C01824=1209.441,-97.315,-38.143,179.366,5.454,149.145
C01825=1209.446,-97.564,-38.133,179.364,5.455,149.146
C01826=1209.452,-97.814,-38.123,179.362,5.454,149.146
C01827=1209.457,-98.064,-38.112,179.360,5.454,149.147
C01828=1209.462,-98.314,-38.102,179.357,5.454,149.148
C01829=1209.467,-98.564,-38.092,179.355,5.454,149.149
C01830=1209.472,-98.813,-38.082,179.353,5.454,149.149
C01831=1209.478,-99.063,-38.071,179.351,5.454,149.150
C01832=1209.483,-99.313,-38.061,179.348,5.453,149.150
C01833=1209.488,-99.562,-38.051,179.346,5.454,149.151
C01834=1209.493,-99.812,-38.041,179.343,5.453,149.152
C01835=1209.498,-100.062,-38.031,179.342,5.453,149.152
C01836=1209.504,-100.311,-38.020,179.339,5.453,149.153
C01837=1209.510,-100.561,-38.010,179.337,5.453,149.154
C01838=1209.515,-100.832,-37.999,179.334,5.453,149.155
C01839=1209.521,-101.104,-37.988,179.331,5.453,149.155
C01840=1209.526,-101.375,-37.977,179.329,5.453,149.156
C01841=1209.532,-101.646,-37.966,179.327,5.453,149.157
C01842=1209.537,-101.896,-37.956,179.325,5.453,149.157
C01843=1209.542,-102.146,-37.945,179.322,5.452,149.158
C01844=1209.548,-102.395,-37.935,179.320,5.452,149.159
C01845=1209.553,-102.645,-37.925,179.318,5.452,149.159
C01846=1209.558,-102.895,-37.915,179.315,5.452,149.160
C01847=1209.564,-103.145,-37.905,179.313,5.452,149.161
C01848=1209.569,-103.395,-37.895,179.311,5.452,149.161
C01849=1209.574,-103.645,-37.885,179.309,5.452,149.162
C01850=1209.579,-103.894,-37.875,179.306,5.452,149.163
C01851=1209.585,-104.143,-37.865,179.304,5.452,149.163
C01852=1209.590,-104.394,-37.854,179.302,5.452,149.164
C01853=1209.594,-104.643,-37.845,179.299,5.451,149.165
C01854=1209.600,-104.892,-37.834,179.297,5.452,149.165
C01855=1209.605,-105.143,-37.825,179.295,5.451,149.166
C01856=1209.611,-105.393,-37.814,179.293,5.451,149.167
C01857=1209.616,-105.642,-37.805,179.290,5.451,149.167
C01858=1209.621,-105.892,-37.795,179.288,5.451,149.168
C01859=1209.626,-106.142,-37.784,179.286,5.451,149.169
C01860=1209.631,-106.391,-37.774,179.284,5.451,149.169
C01861=1209.637,-106.641,-37.765,179.281,5.450,149.170
C01862=1209.642,-106.891,-37.754,179.279,5.451,149.171
C01863=1209.647,-107.141,-37.745,179.277,5.450,149.171
C01864=1209.653,-107.390,-37.734,179.275,5.451,149.172
C01865=1209.658,-107.640,-37.724,179.272,5.450,149.172
C01866=1209.663,-107.890,-37.715,179.270,5.450,149.173
C01867=1209.668,-108.140,-37.705,179.268,5.450,149.174
C01868=1209.674,-108.389,-37.695,179.265,5.450,149.175
C01869=1209.679,-108.639,-37.685,179.263,5.449,149.175
C01870=1209.684,-108.889,-37.675,179.261,5.450,149.176
C01871=1209.689,-109.139,-37.665,179.259,5.449,149.176
C01872=1209.695,-109.388,-37.655,179.256,5.450,149.177
C01873=1209.700,-109.638,-37.645,179.254,5.449,149.178
C01874=1209.705,-109.888,-37.636,179.252,5.449,149.178
C01875=1209.710,-110.138,-37.626,179.249,5.449,149.179
C01876=1209.716,-110.387,-37.615,179.247,5.449,149.180
C01877=1209.721,-110.637,-37.606,179.245,5.448,149.180
C01878=1209.727,-110.887,-37.596,179.243,5.449,149.181
C01879=1209.732,-111.136,-37.587,179.240,5.448,149.182
C01880=1209.737,-111.386,-37.576,179.238,5.449,149.182
C01881=1209.743,-111.636,-37.567,179.236,5.448,149.183
C01882=1209.747,-111.886,-37.557,179.234,5.448,149.184
C01883=1209.753,-112.135,-37.547,179.231,5.448,149.184
C01884=1209.758,-112.385,-37.538,179.229,5.448,149.185
C01885=1209.763,-112.635,-37.527,179.228,5.448,149.186
C01886=1209.768,-112.885,-37.518,179.225,5.448,149.186
C01887=1209.774,-113.135,-37.508,179.223,5.448,149.187
C01888=1209.780,-113.384,-37.498,179.220,5.448,149.188
C01889=1209.785,-113.634,-37.489,179.219,5.448,149.188
C01890=1209.790,-113.884,-37.479,179.216,5.448,149.189
C01891=1209.795,-114.134,-37.469,179.214,5.448,149.190
C01892=1209.800,-114.384,-37.459,179.212,5.447,149.190
C01893=1209.805,-114.633,-37.450,179.210,5.448,149.191
C01894=1209.811,-114.883,-37.440,179.207,5.447,149.192
C01895=1209.816,-115.132,-37.431,179.205,5.448,149.192
C01896=1209.822,-115.382,-37.420,179.203,5.447,149.193
C01897=1209.826,-115.633,-37.411,179.201,5.447,149.193
C01898=1209.832,-115.882,-37.401,179.198,5.447,149.194
C01899=1209.837,-116.132,-37.392,179.196,5.447,149.195
C01900=1209.843,-116.381,-37.382,179.194,5.446,149.195
C01901=1209.848,-116.631,-37.373,179.192,5.447,149.196
C01902=1209.853,-116.881,-37.363,179.189,5.446,149.197
C01903=1209.858,-117.130,-37.353,179.187,5.446,149.197
C01904=1209.864,-117.381,-37.343,179.185,5.446,149.198
C01905=1209.868,-117.630,-37.334,179.182,5.446,149.199
C01906=1209.874,-117.880,-37.324,179.180,5.447,149.199
C01907=1209.879,-118.130,-37.315,179.178,5.446,149.200
C01908=1209.885,-118.380,-37.305,179.176,5.446,149.201
C01909=1209.890,-118.629,-37.296,179.173,5.446,149.201
C01910=1209.895,-118.879,-37.287,179.172,5.446,149.202
C01911=1209.901,-119.128,-37.276,179.169,5.445,149.203
C01912=1209.906,-119.378,-37.268,179.167,5.446,149.203
C01913=1209.911,-119.628,-37.257,179.164,5.445,149.204
C01914=1209.916,-119.878,-37.248,179.163,5.445,149.204
C01915=1209.922,-120.128,-37.239,179.160,5.445,149.205
C01916=1209.927,-120.378,-37.229,179.158,5.445,149.206
C01917=1209.932,-120.628,-37.220,179.156,5.445,149.206
C01918=1209.938,-120.877,-37.210,179.154,5.445,149.207
C01919=1209.943,-121.127,-37.201,179.151,5.445,149.208
C01920=1209.948,-121.376,-37.191,179.149,5.445,149.208
C01921=1209.953,-121.626,-37.182,179.147,5.445,149.209
C01922=1209.959,-121.876,-37.173,179.145,5.445,149.210
C01923=1209.964,-122.126,-37.163,179.143,5.445,149.210
C01924=1209.969,-122.376,-37.154,179.140,5.444,149.211
C01925=1209.974,-122.625,-37.144,179.138,5.445,149.212
C01926=1209.980,-122.875,-37.135,179.136,5.444,149.212
C01927=1209.985,-123.126,-37.125,179.134,5.444,149.213
C01928=1209.990,-123.375,-37.115,179.131,5.444,149.214
C01929=1209.996,-123.625,-37.106,179.129,5.444,149.214
C01930=1210.000,-123.874,-37.097,179.127,5.443,149.215
C01931=1210.006,-124.124,-37.087,179.125,5.444,149.216
C01932=1210.011,-124.374,-37.078,179.122,5.443,149.216
C01933=1210.016,-124.623,-37.069,179.121,5.443,149.217
C01934=1210.022,-124.874,-37.059,179.119,5.444,149.217
C01935=1210.027,-125.123,-37.050,179.116,5.443,149.218
C01936=1210.032,-125.373,-37.041,179.114,5.444,149.219
C01937=1210.038,-125.623,-37.031,179.112,5.443,149.219
C01938=1210.043,-125.873,-37.022,179.110,5.443,149.220
C01939=1210.048,-126.123,-37.013,179.107,5.443,149.221
C01940=1210.054,-126.372,-37.003,179.105,5.443,149.221
C01941=1210.059,-126.622,-36.994,179.103,5.443,149.222
C01942=1209.638,-126.632,-37.032,179.099,5.446,149.224
C01943=1209.632,-126.382,-37.041,179.101,5.447,149.223
C01944=1209.628,-126.133,-37.051,179.103,5.446,149.223
C01945=1209.622,-125.883,-37.060,179.106,5.447,149.222
C01946=1209.617,-125.633,-37.069,179.107,5.447,149.221
C01947=1209.611,-125.383,-37.078,179.110,5.447,149.221
C01948=1209.606,-125.134,-37.088,179.112,5.447,149.220
C01949=1209.601,-124.884,-37.097,179.114,5.447,149.220
C01950=1209.595,-124.634,-37.106,179.116,5.447,149.219
C01951=1209.590,-124.385,-37.116,179.118,5.447,149.218
C01952=1209.585,-124.135,-37.125,179.121,5.447,149.218
C01953=1209.580,-123.885,-37.134,179.123,5.447,149.217
C01954=1209.574,-123.635,-37.144,179.125,5.447,149.216
C01955=1209.569,-123.385,-37.153,179.127,5.447,149.215
C01956=1209.564,-123.136,-37.162,179.130,5.448,149.215
C01957=1209.558,-122.886,-37.172,179.132,5.447,149.214
C01958=1209.553,-122.636,-37.181,179.134,5.448,149.214
C01959=1209.548,-122.387,-37.191,179.136,5.448,149.213
C01960=1209.542,-122.137,-37.200,179.139,5.448,149.212
C01961=1209.537,-121.887,-37.209,179.141,5.448,149.212
C01962=1209.532,-121.638,-37.219,179.143,5.449,149.211
C01963=1209.526,-121.388,-37.228,179.145,5.448,149.210
C01964=1209.521,-121.138,-37.238,179.147,5.448,149.210
C01965=1209.516,-120.887,-37.248,179.149,5.449,149.209
C01966=1209.511,-120.638,-37.257,179.151,5.448,149.209
C01967=1209.506,-120.388,-37.266,179.154,5.449,149.208
C01968=1209.500,-120.138,-37.276,179.156,5.448,149.207
C01969=1209.495,-119.889,-37.285,179.158,5.449,149.207
C01970=1209.489,-119.639,-37.295,179.160,5.449,149.206
C01971=1209.484,-119.390,-37.305,179.163,5.449,149.205
C01972=1209.479,-119.139,-37.314,179.165,5.449,149.205
C01973=1209.474,-118.890,-37.324,179.167,5.449,149.204
C01974=1209.468,-118.640,-37.333,179.169,5.449,149.203
C01975=1209.463,-118.391,-37.343,179.172,5.449,149.203
C01976=1209.458,-118.140,-37.352,179.174,5.449,149.202
C01977=1209.453,-117.891,-37.362,179.176,5.450,149.201
C01978=1209.448,-117.641,-37.371,179.179,5.449,149.201
C01979=1209.442,-117.391,-37.381,179.180,5.449,149.200
C01980=1209.437,-117.141,-37.390,179.183,5.450,149.199
C01981=1209.431,-116.892,-37.400,179.185,5.449,149.199
C01982=1209.426,-116.642,-37.409,179.188,5.450,149.198
C01983=1209.420,-116.392,-37.420,179.189,5.450,149.197
C01984=1209.416,-116.142,-37.429,179.192,5.450,149.197
C01985=1209.410,-115.892,-37.439,179.194,5.450,149.196
C01986=1209.405,-115.643,-37.448,179.196,5.451,149.196
C01987=1209.399,-115.393,-37.458,179.198,5.450,149.195
C01988=1209.395,-115.144,-37.468,179.201,5.451,149.194
C01989=1209.389,-114.894,-37.477,179.203,5.450,149.193
C01990=1209.384,-114.644,-37.487,179.205,5.451,149.193
C01991=1209.379,-114.394,-37.497,179.207,5.451,149.192
C01992=1209.374,-114.144,-37.506,179.210,5.451,149.191
C01993=1209.368,-113.895,-37.517,179.212,5.451,149.191
C01994=1209.363,-113.645,-37.525,179.214,5.452,149.190
C01995=1209.357,-113.395,-37.536,179.216,5.451,149.190
C01996=1209.352,-113.145,-37.545,179.219,5.452,149.189
C01997=1209.347,-112.895,-37.555,179.221,5.452,149.188
C01998=1209.342,-112.646,-37.565,179.223,5.452,149.188
C01999=1209.336,-112.396,-37.574,179.225,5.452,149.187
C02000=1209.331,-112.146,-37.584,179.228,5.452,149.186
C02001=1209.326,-111.897,-37.594,179.230,5.452,149.186
C02002=1209.320,-111.647,-37.604,179.232,5.452,149.185
C02003=1209.316,-111.397,-37.614,179.234,5.452,149.184
C02004=1209.310,-111.147,-37.624,179.237,5.452,149.184
C02005=1209.305,-110.898,-37.633,179.239,5.452,149.183
C02006=1209.299,-110.648,-37.643,179.241,5.452,149.182
C02007=1209.294,-110.399,-37.653,179.243,5.452,149.182
C02008=1209.289,-110.148,-37.662,179.245,5.452,149.181
C02009=1209.284,-109.898,-37.673,179.248,5.453,149.181
C02010=1209.279,-109.649,-37.682,179.250,5.452,149.180
C02011=1209.273,-109.400,-37.692,179.253,5.453,149.179
C02012=1209.268,-109.149,-37.702,179.254,5.453,149.179
C02013=1209.263,-108.900,-37.712,179.257,5.453,149.178
C02014=1209.257,-108.650,-37.722,179.259,5.453,149.177
C02015=1209.252,-108.400,-37.732,179.262,5.453,149.176
C02016=1209.247,-108.151,-37.741,179.263,5.453,149.176
C02017=1209.242,-107.900,-37.752,179.266,5.454,149.175
C02018=1209.236,-107.651,-37.762,179.268,5.453,149.175
C02019=1209.231,-107.402,-37.772,179.271,5.454,149.174
C02020=1209.225,-107.151,-37.781,179.272,5.454,149.173
C02021=1209.220,-106.901,-37.792,179.275,5.454,149.173
C02022=1209.215,-106.652,-37.801,179.277,5.454,149.172
C02023=1209.210,-106.402,-37.811,179.280,5.454,149.171
C02024=1209.205,-106.152,-37.822,179.281,5.454,149.171
C02025=1209.200,-105.902,-37.831,179.284,5.455,149.170
C02026=1209.194,-105.653,-37.841,179.286,5.454,149.169
C02027=1209.189,-105.403,-37.851,179.289,5.455,149.169
C02028=1209.184,-105.153,-37.861,179.291,5.454,149.168
C02029=1209.179,-104.904,-37.872,179.293,5.455,149.167
C02030=1209.173,-104.654,-37.882,179.295,5.455,149.167
C02031=1209.168,-104.405,-37.891,179.298,5.455,149.166
C02032=1209.163,-104.154,-37.901,179.300,5.455,149.165
C02033=1209.157,-103.905,-37.911,179.302,5.456,149.165
C02034=1209.152,-103.655,-37.922,179.304,5.455,149.164
C02035=1209.147,-103.405,-37.932,179.307,5.456,149.163
C02036=1209.142,-103.156,-37.942,179.309,5.455,149.163
C02037=1209.136,-102.906,-37.952,179.311,5.456,149.162
C02038=1209.132,-102.656,-37.962,179.313,5.456,149.161
C02039=1209.126,-102.407,-37.972,179.316,5.456,149.161
C02040=1209.121,-102.157,-37.982,179.318,5.456,149.160
C02041=1209.115,-101.906,-37.992,179.320,5.456,149.159
C02042=1209.111,-101.657,-38.002,179.322,5.456,149.159
C02043=1209.105,-101.385,-38.013,179.325,5.456,149.158
C02044=1209.099,-101.115,-38.024,179.328,5.457,149.157
C02045=1209.093,-100.843,-38.036,179.330,5.457,149.157
C02046=1209.088,-100.572,-38.046,179.332,5.457,149.156
C02047=1209.082,-100.322,-38.057,179.334,5.457,149.155
C02048=1209.077,-100.073,-38.067,179.337,5.457,149.154
C02049=1209.072,-99.822,-38.077,179.339,5.457,149.154
C02050=1209.067,-99.573,-38.087,179.341,5.457,149.153
C02051=1209.062,-99.323,-38.098,179.343,5.457,149.153
C02052=1209.056,-99.073,-38.108,179.346,5.457,149.152
C02053=1209.051,-98.824,-38.118,179.348,5.457,149.151
C02054=1209.046,-98.574,-38.129,179.351,5.457,149.150
C02055=1209.041,-98.324,-38.138,179.352,5.457,149.150
C02056=1209.035,-98.075,-38.148,179.355,5.458,149.149
C02057=1209.030,-97.825,-38.159,179.357,5.458,149.149
C02058=1209.024,-97.575,-38.169,179.360,5.458,149.148
C02059=1209.019,-97.326,-38.179,179.361,5.458,149.147
C02060=1209.014,-97.075,-38.190,179.364,5.458,149.147
C02061=1209.008,-96.826,-38.200,179.366,5.458,149.146
C02062=1209.004,-96.576,-38.210,179.369,5.458,149.145
C02063=1208.999,-96.327,-38.221,179.372,5.459,149.144
C02064=1208.993,-96.077,-38.231,179.373,5.459,149.144
C02065=1208.988,-95.827,-38.242,179.376,5.459,149.143
C02066=1208.983,-95.578,-38.252,179.378,5.459,149.143
C02067=1208.978,-95.327,-38.263,179.381,5.459,149.142
C02068=1208.972,-95.078,-38.273,179.383,5.459,149.141
C02069=1208.966,-94.828,-38.283,179.385,5.460,149.141
C02070=1208.961,-94.578,-38.294,179.387,5.459,149.140
C02071=1208.956,-94.328,-38.304,179.390,5.460,149.139
C02072=1208.952,-94.079,-38.315,179.392,5.459,149.139
C02073=1208.946,-93.830,-38.325,179.394,5.460,149.138
C02074=1208.941,-93.579,-38.335,179.396,5.460,149.137
C02075=1208.936,-93.330,-38.346,179.399,5.460,149.137
C02076=1208.930,-93.080,-38.356,179.401,5.460,149.136
C02077=1208.925,-92.830,-38.366,179.403,5.460,149.135
C02078=1208.919,-92.580,-38.377,179.406,5.460,149.135
C02079=1208.915,-92.331,-38.388,179.408,5.461,149.134
C02080=1208.909,-92.081,-38.398,179.410,5.460,149.133
C02081=1208.904,-91.831,-38.409,179.413,5.461,149.133
C02082=1208.899,-91.581,-38.419,179.415,5.460,149.132
C02083=1208.894,-91.331,-38.429,179.417,5.461,149.131
C02084=1208.888,-91.082,-38.440,179.419,5.462,149.131
C02085=1208.883,-90.833,-38.451,179.422,5.461,149.130
C02086=1208.878,-90.583,-38.461,179.424,5.462,149.129
C02087=1208.872,-90.333,-38.471,179.426,5.461,149.129
C02088=1208.867,-90.083,-38.483,179.429,5.462,149.128
C02089=1208.862,-89.834,-38.493,179.431,5.462,149.127
C02090=1208.857,-89.584,-38.503,179.433,5.462,149.127
C02091=1208.851,-89.334,-38.514,179.435,5.462,149.126
C02092=1208.846,-89.084,-38.525,179.438,5.462,149.125
C02093=1208.841,-88.835,-38.535,179.440,5.462,149.125
C02094=1208.836,-88.585,-38.546,179.442,5.463,149.124
C02095=1208.831,-88.336,-38.557,179.444,5.462,149.123
C02096=1208.826,-88.085,-38.567,179.447,5.463,149.123
C02097=1208.820,-87.836,-38.577,179.449,5.462,149.122
C02098=1208.815,-87.586,-38.589,179.452,5.463,149.121
C02099=1208.810,-87.337,-38.599,179.454,5.463,149.120
C02100=1208.805,-87.086,-38.609,179.456,5.463,149.120
C02101=1208.799,-86.837,-38.620,179.459,5.464,149.119
C02102=1208.794,-86.587,-38.631,179.461,5.463,149.119
C02103=1208.789,-86.338,-38.641,179.464,5.464,149.118
C02104=1208.784,-86.088,-38.652,179.466,5.463,149.117
C02105=1208.779,-85.838,-38.663,179.468,5.464,149.117
C02106=1208.774,-85.588,-38.673,179.470,5.464,149.116
C02107=1208.769,-85.339,-38.685,179.473,5.464,149.115
C02108=1208.762,-85.089,-38.695,179.475,5.464,149.115
C02109=1208.757,-84.839,-38.706,179.477,5.464,149.114
C02110=1208.752,-84.590,-38.717,179.479,5.464,149.113
C02111=1208.747,-84.339,-38.727,179.482,5.465,149.113
C02112=1208.742,-84.091,-38.738,179.484,5.465,149.112
C02113=1208.737,-83.840,-38.749,179.486,5.465,149.111
C02114=1208.732,-83.591,-38.760,179.489,5.465,149.111
C02115=1208.727,-83.341,-38.770,179.491,5.465,149.110
C02116=1208.722,-83.091,-38.781,179.494,5.465,149.109
C02117=1208.716,-82.842,-38.793,179.495,5.465,149.109
C02118=1208.711,-82.591,-38.803,179.498,5.466,149.108
C02119=1208.705,-82.342,-38.814,179.500,5.465,149.107
C02120=1208.700,-82.092,-38.825,179.503,5.466,149.106
C02121=1208.696,-81.843,-38.836,179.505,5.466,149.106
C02122=1208.690,-81.593,-38.846,179.507,5.466,149.105
C02123=1208.685,-81.343,-38.857,179.510,5.467,149.105
C02124=1208.679,-81.094,-38.868,179.512,5.466,149.104
C02125=1208.674,-80.844,-38.879,179.515,5.467,149.103
C02126=1208.669,-80.594,-38.890,179.517,5.466,149.102
C02127=1208.664,-80.345,-38.901,179.519,5.467,149.102
C02128=1208.659,-80.095,-38.912,179.521,5.467,149.101
C02129=1208.653,-79.845,-38.923,179.524,5.467,149.101
C02130=1208.648,-79.595,-38.934,179.526,5.468,149.100
C02131=1208.643,-79.345,-38.945,179.528,5.467,149.099
C02132=1208.638,-79.096,-38.955,179.531,5.468,149.098
C02133=1208.633,-78.846,-38.966,179.533,5.467,149.098
C02134=1208.627,-78.597,-38.978,179.535,5.468,149.097
C02135=1208.622,-78.347,-38.989,179.537,5.468,149.097
C02136=1208.617,-78.097,-39.000,179.540,5.468,149.096
C02137=1208.612,-77.848,-39.010,179.542,5.468,149.095
C02138=1208.606,-77.598,-39.022,179.545,5.468,149.094
C02139=1208.601,-77.347,-39.032,179.547,5.469,149.094
C02140=1208.596,-77.099,-39.043,179.549,5.468,149.093
C02141=1208.591,-76.849,-39.055,179.552,5.469,149.093
C02142=1208.586,-76.598,-39.066,179.554,5.469,149.092
C02143=1208.580,-76.349,-39.077,179.556,5.469,149.091
C02144=1208.576,-76.100,-39.088,179.559,5.469,149.090
C02145=1208.570,-75.849,-39.099,179.561,5.469,149.090
C02146=1208.565,-75.600,-39.110,179.564,5.470,149.089
C02147=1208.559,-75.329,-39.122,179.566,5.470,149.088
C02148=1208.554,-75.059,-39.134,179.569,5.470,149.088
C02149=1208.548,-74.788,-39.146,179.571,5.470,149.087
C02150=1208.542,-74.517,-39.158,179.573,5.470,149.086
C02151=1208.537,-74.268,-39.169,179.576,5.470,149.085
C02152=1208.531,-74.018,-39.180,179.579,5.471,149.085
C02153=1208.526,-73.768,-39.192,179.580,5.471,149.084
C02154=1208.522,-73.519,-39.203,179.583,5.471,149.084
C02155=1208.516,-73.269,-39.214,179.585,5.471,149.083
C02156=1208.511,-73.019,-39.225,179.588,5.471,149.082
C02157=1208.506,-72.770,-39.236,179.590,5.471,149.081
C02158=1208.500,-72.520,-39.248,179.593,5.472,149.081
C02159=1208.495,-72.271,-39.259,179.595,5.472,149.080
C02160=1208.490,-72.020,-39.270,179.597,5.472,149.080
C02161=1208.484,-71.771,-39.281,179.599,5.472,149.079
C02162=1208.480,-71.522,-39.292,179.602,5.472,149.078
C02163=1208.475,-71.272,-39.304,179.604,5.473,149.077
C02164=1208.469,-71.021,-39.315,179.607,5.473,149.077
C02165=1208.464,-70.773,-39.326,179.609,5.473,149.076
C02166=1208.458,-70.523,-39.338,179.611,5.473,149.076
C02167=1208.454,-70.273,-39.349,179.613,5.473,149.075
C02168=1208.449,-70.023,-39.360,179.616,5.473,149.074
C02169=1208.443,-69.773,-39.371,179.618,5.473,149.073
C02170=1208.438,-69.524,-39.382,179.621,5.474,149.073
C02171=1208.433,-69.274,-39.394,179.623,5.474,149.072
C02172=1208.428,-69.024,-39.406,179.625,5.474,149.071
C02173=1208.423,-68.775,-39.417,179.628,5.474,149.071
C02174=1208.417,-68.525,-39.428,179.630,5.474,149.070
C02175=1208.412,-68.275,-39.439,179.632,5.475,149.069
C02176=1208.407,-68.025,-39.451,179.635,5.475,149.069
C02177=1208.401,-67.776,-39.462,179.637,5.475,149.068
C02178=1208.396,-67.526,-39.474,179.640,5.475,149.067
C02179=1208.391,-67.277,-39.485,179.642,5.475,149.067
C02180=1208.386,-67.027,-39.497,179.644,5.476,149.066
C02181=1208.381,-66.777,-39.508,179.647,5.476,149.065
C02182=1208.375,-66.528,-39.520,179.649,5.476,149.065
C02183=1208.370,-66.278,-39.530,179.651,5.476,149.064
C02184=1208.366,-66.028,-39.542,179.654,5.476,149.063
C02185=1208.360,-65.778,-39.553,179.656,5.476,149.063
C02186=1208.355,-65.529,-39.565,179.659,5.477,149.062
C02187=1208.349,-65.279,-39.576,179.661,5.476,149.061
C02188=1208.345,-65.030,-39.588,179.663,5.477,149.061
C02189=1208.339,-64.780,-39.599,179.665,5.477,149.060
C02190=1208.335,-64.530,-39.611,179.668,5.477,149.059
C02191=1208.329,-64.280,-39.623,179.671,5.478,149.059
C02192=1208.324,-64.031,-39.633,179.673,5.477,149.058
C02193=1208.318,-63.781,-39.645,179.675,5.478,149.057
C02194=1208.313,-63.531,-39.657,179.677,5.477,149.056
C02195=1208.308,-63.282,-39.669,179.680,5.478,149.056
C02196=1208.303,-63.032,-39.680,179.682,5.479,149.055
C02197=1208.298,-62.782,-39.692,179.684,5.478,149.055
C02198=1208.293,-62.532,-39.704,179.687,5.479,149.054
C02199=1208.287,-62.283,-39.715,179.689,5.478,149.053
C02200=1208.282,-62.033,-39.726,179.692,5.479,149.052
C02201=1208.277,-61.784,-39.738,179.694,5.479,149.052
C02202=1208.272,-61.534,-39.750,179.697,5.479,149.051
C02203=1208.267,-61.284,-39.761,179.699,5.480,149.051
C02204=1208.262,-61.034,-39.773,179.701,5.479,149.050
C02205=1208.256,-60.784,-39.785,179.703,5.480,149.049
C02206=1208.251,-60.535,-39.796,179.706,5.480,149.048
C02207=1208.246,-60.285,-39.807,179.708,5.480,149.048
C02208=1208.241,-60.036,-39.819,179.711,5.480,149.047
C02209=1208.236,-59.787,-39.831,179.714,5.481,149.046
C02210=1208.230,-59.537,-39.843,179.715,5.481,149.046
C02211=1208.226,-59.287,-39.855,179.718,5.481,149.045
C02212=1208.220,-59.037,-39.866,179.720,5.481,149.044
C02213=1208.216,-58.787,-39.878,179.723,5.481,149.044
C02214=1208.210,-58.537,-39.890,179.725,5.482,149.043
C02215=1208.205,-58.287,-39.901,179.727,5.482,149.042
C02216=1208.200,-58.039,-39.913,179.730,5.482,149.042
C02217=1208.194,-57.789,-39.925,179.732,5.482,149.041
C02218=1208.189,-57.539,-39.937,179.734,5.482,149.040
C02219=1208.184,-57.290,-39.948,179.737,5.483,149.040
C02220=1208.179,-57.040,-39.960,179.739,5.483,149.039
C02221=1208.173,-56.790,-39.972,179.742,5.483,149.038
C02222=1208.169,-56.541,-39.984,179.744,5.483,149.038
C02223=1208.164,-56.291,-39.996,179.746,5.483,149.037
C02224=1208.158,-56.041,-40.008,179.749,5.484,149.036
C02225=1208.153,-55.791,-40.019,179.751,5.483,149.035
C02226=1208.148,-55.541,-40.031,179.753,5.484,149.035
C02227=1208.143,-55.292,-40.044,179.756,5.485,149.034
C02228=1208.138,-55.042,-40.055,179.758,5.484,149.034
C02229=1208.133,-54.793,-40.067,179.761,5.485,149.033
C02230=1208.127,-54.543,-40.079,179.763,5.485,149.032
C02231=1208.123,-54.294,-40.091,179.765,5.485,149.031
C02232=1208.117,-54.044,-40.102,179.768,5.485,149.031
C02233=1208.112,-53.794,-40.114,179.771,5.486,149.030
C02234=1208.107,-53.544,-40.127,179.772,5.486,149.030
C02235=1208.102,-53.295,-40.138,179.775,5.486,149.029
C02236=1208.097,-53.045,-40.150,179.777,5.486,149.028
C02237=1208.091,-52.795,-40.162,179.780,5.486,149.027
C02238=1208.086,-52.546,-40.175,179.782,5.487,149.027
C02239=1208.081,-52.297,-40.186,179.785,5.486,149.026
C02240=1208.076,-52.047,-40.197,179.787,5.487,149.025
C02241=1208.070,-51.797,-40.210,179.790,5.487,149.025
C02242=1208.065,-51.547,-40.222,179.792,5.487,149.024
C02243=1208.060,-51.298,-40.233,179.794,5.488,149.023
C02244=1208.056,-51.048,-40.246,179.797,5.488,149.023
C02245=1208.050,-50.798,-40.258,179.799,5.488,149.022
C02246=1208.045,-50.548,-40.270,179.802,5.488,149.021
C02247=1208.040,-50.299,-40.283,179.804,5.489,149.021
C02248=1208.035,-50.049,-40.294,179.806,5.488,149.020
C02249=1208.030,-49.800,-40.306,179.809,5.489,149.019
C02250=1208.025,-49.550,-40.318,179.811,5.489,149.019
C02251=1208.019,-49.280,-40.331,179.814,5.489,149.018
C02252=1208.013,-49.010,-40.344,179.816,5.489,149.017
C02253=1208.008,-48.740,-40.358,179.819,5.490,149.016
C02254=1208.002,-48.470,-40.371,179.822,5.490,149.016
C02255=1207.996,-48.220,-40.383,179.824,5.490,149.015
C02256=1207.992,-47.971,-40.395,179.827,5.490,149.014
C02257=1207.986,-47.721,-40.407,179.829,5.491,149.014
C02258=1207.981,-47.472,-40.419,179.831,5.491,149.013
C02259=1207.976,-47.222,-40.431,179.833,5.491,149.012
C02260=1207.971,-46.973,-40.444,179.836,5.492,149.012
C02261=1207.966,-46.722,-40.456,179.838,5.492,149.011
C02262=1207.961,-46.473,-40.468,179.841,5.492,149.010
C02263=1207.956,-46.223,-40.480,179.844,5.492,149.010
C02264=1207.951,-45.974,-40.492,179.846,5.492,149.009
C02265=1207.946,-45.724,-40.504,179.848,5.493,149.008
C02266=1207.940,-45.474,-40.517,179.851,5.493,149.008
C02267=1207.935,-45.224,-40.529,179.853,5.493,149.007
C02268=1207.930,-44.975,-40.541,179.855,5.494,149.006
C02269=1207.924,-44.725,-40.553,179.858,5.494,149.006
C02270=1207.919,-44.476,-40.566,179.860,5.494,149.005
C02271=1207.914,-44.226,-40.578,179.863,5.494,149.004
C02272=1207.909,-43.976,-40.591,179.865,5.495,149.004
C02273=1207.904,-43.726,-40.603,179.867,5.494,149.003
C02274=1207.899,-43.477,-40.615,179.870,5.495,149.002
C02275=1207.894,-43.227,-40.628,179.873,5.495,149.001
C02276=1207.888,-42.977,-40.640,179.875,5.495,149.001
C02277=1207.884,-42.728,-40.652,179.877,5.496,149.000
C02278=1207.878,-42.479,-40.664,179.880,5.496,149.000
C02279=1207.873,-42.229,-40.676,179.882,5.496,148.999
C02280=1207.868,-41.980,-40.689,179.884,5.496,148.998
C02281=1207.863,-41.729,-40.701,179.887,5.497,148.997
C02282=1207.858,-41.480,-40.714,179.889,5.496,148.997
C02283=1207.853,-41.230,-40.725,179.892,5.497,148.996
C02284=1207.848,-40.981,-40.738,179.894,5.497,148.995
C02285=1207.843,-40.731,-40.751,179.896,5.497,148.995
C02286=1207.837,-40.481,-40.763,179.899,5.498,148.994
C02287=1207.833,-40.231,-40.776,179.901,5.498,148.994
C02288=1207.827,-39.982,-40.788,179.903,5.498,148.993
C02289=1207.822,-39.732,-40.800,179.906,5.498,148.992
C02290=1207.817,-39.483,-40.813,179.909,5.499,148.991
C02291=1207.812,-39.234,-40.825,179.911,5.499,148.991
C02292=1207.806,-38.984,-40.838,179.913,5.499,148.990
C02293=1207.801,-38.733,-40.851,179.916,5.500,148.989
C02294=1207.796,-38.484,-40.863,179.918,5.500,148.989
C02295=1207.791,-38.235,-40.876,179.920,5.500,148.988
C02296=1207.785,-37.985,-40.888,179.923,5.500,148.987
C02297=1207.780,-37.735,-40.900,179.926,5.501,148.987
C02298=1207.775,-37.486,-40.913,179.928,5.501,148.986
C02299=1207.771,-37.236,-40.926,179.930,5.501,148.985
C02300=1207.765,-36.986,-40.938,179.933,5.502,148.985
C02301=1207.760,-36.737,-40.950,179.935,5.501,148.984
C02302=1207.755,-36.487,-40.963,179.938,5.502,148.983
C02303=1207.750,-36.237,-40.976,179.941,5.502,148.983
C02304=1207.745,-35.988,-40.989,179.942,5.502,148.982
C02305=1207.739,-35.738,-41.001,179.945,5.503,148.981
C02306=1207.734,-35.489,-41.014,179.947,5.503,148.981
C02307=1207.729,-35.239,-41.026,179.950,5.503,148.980
C02308=1207.724,-34.989,-41.039,179.952,5.503,148.979
C02309=1207.719,-34.740,-41.052,179.955,5.504,148.979
C02310=1207.714,-34.490,-41.064,179.958,5.504,148.978
C02311=1207.709,-34.241,-41.076,179.960,5.504,148.977
C02312=1207.703,-33.990,-41.090,179.962,5.504,148.976
C02313=1207.698,-33.741,-41.102,179.964,5.505,148.976
C02314=1207.693,-33.492,-41.115,179.966,5.505,148.975
C02315=1207.688,-33.242,-41.128,179.969,5.505,148.975
C02316=1207.684,-32.992,-41.141,179.972,5.506,148.974
C02317=1207.678,-32.743,-41.153,179.974,5.506,148.973
C02318=1207.672,-32.493,-41.166,179.977,5.506,148.973
C02319=1207.667,-32.243,-41.178,179.979,5.506,148.972
C02320=1207.663,-31.993,-41.191,179.982,5.507,148.971
C02321=1207.657,-31.744,-41.204,179.984,5.507,148.970
C02322=1207.652,-31.495,-41.216,179.986,5.507,148.970
C02323=1207.647,-31.244,-41.230,179.989,5.508,148.969
C02324=1207.642,-30.995,-41.243,179.991,5.508,148.969
C02325=1207.637,-30.746,-41.255,179.994,5.508,148.968
C02326=1207.632,-30.497,-41.268,179.996,5.509,148.967
C02327=1207.627,-30.246,-41.281,179.999,5.509,148.966
C02328=1207.621,-29.997,-41.294,-179.999,5.509,148.966
C02329=1207.616,-29.748,-41.307,-179.996,5.509,148.965
C02330=1207.612,-29.498,-41.320,-179.994,5.510,148.964
C02331=1207.607,-29.248,-41.332,-179.992,5.510,148.964
C02332=1207.601,-28.999,-41.345,-179.989,5.510,148.963
C02333=1207.596,-28.749,-41.358,-179.987,5.511,148.963
C02334=1207.591,-28.499,-41.371,-179.984,5.511,148.962
C02335=1207.586,-28.250,-41.384,-179.982,5.511,148.961
C02336=1207.581,-28.000,-41.397,-179.979,5.511,148.960
C02337=1207.576,-27.750,-41.410,-179.977,5.512,148.960
C02338=1207.570,-27.501,-41.422,-179.974,5.512,148.959
C02339=1207.565,-27.251,-41.436,-179.972,5.512,148.958
C02340=1207.560,-27.001,-41.448,-179.970,5.513,148.958
C02341=1207.555,-26.752,-41.461,-179.967,5.513,148.957
C02342=1207.550,-26.502,-41.474,-179.965,5.514,148.956
C02343=1207.545,-26.252,-41.487,-179.962,5.513,148.956
C02344=1207.540,-26.004,-41.501,-179.960,5.514,148.955
C02345=1207.535,-25.754,-41.514,-179.957,5.514,148.954
C02346=1207.529,-25.504,-41.527,-179.955,5.514,148.954
C02347=1207.525,-25.254,-41.540,-179.952,5.514,148.953
C02348=1207.520,-25.005,-41.552,-179.950,5.515,148.952
C02349=1207.514,-24.755,-41.565,-179.948,5.516,148.952
C02350=1207.509,-24.505,-41.578,-179.945,5.515,148.951
C02351=1207.505,-24.256,-41.592,-179.943,5.516,148.950
C02352=1207.499,-24.007,-41.605,-179.940,5.516,148.950
C02353=1207.494,-23.757,-41.618,-179.937,5.517,148.949
C02354=1207.488,-23.507,-41.631,-179.935,5.517,148.948
C02355=1207.483,-23.237,-41.645,-179.933,5.517,148.948
C02356=1207.478,-22.968,-41.660,-179.930,5.518,148.947
C02357=1207.472,-22.699,-41.673,-179.927,5.518,148.946
C02358=1207.466,-22.429,-41.687,-179.925,5.518,148.946
C02359=1207.462,-22.180,-41.701,-179.922,5.519,148.945
C02360=1207.456,-21.930,-41.714,-179.920,5.519,148.944
C02361=1207.451,-21.681,-41.727,-179.917,5.519,148.943
C02362=1207.446,-21.430,-41.740,-179.915,5.520,148.943
C02363=1207.441,-21.181,-41.754,-179.912,5.520,148.942
C02364=1207.437,-20.931,-41.767,-179.910,5.520,148.941
C02365=1207.431,-20.682,-41.780,-179.907,5.520,148.941
C02366=1207.426,-20.433,-41.792,-179.905,5.521,148.940
C02367=1207.421,-20.183,-41.807,-179.902,5.522,148.940
C02368=1207.416,-19.933,-41.819,-179.900,5.521,148.939
C02369=1207.410,-19.683,-41.833,-179.898,5.522,148.938
C02370=1207.405,-19.434,-41.846,-179.895,5.522,148.937
C02371=1207.400,-19.184,-41.860,-179.892,5.523,148.937
C02372=1207.395,-18.935,-41.872,-179.890,5.522,148.936
C02373=1207.390,-18.684,-41.886,-179.888,5.523,148.935
C02374=1207.385,-18.436,-41.899,-179.885,5.523,148.935
C02375=1207.380,-18.185,-41.913,-179.883,5.524,148.934
C02376=1207.375,-17.936,-41.925,-179.880,5.525,148.934
C02377=1207.369,-17.687,-41.939,-179.878,5.524,148.933
C02378=1207.365,-17.437,-41.952,-179.875,5.525,148.932
C02379=1207.359,-17.187,-41.966,-179.873,5.525,148.931
C02380=1207.355,-16.938,-41.979,-179.870,5.526,148.931
C02381=1207.349,-16.688,-41.992,-179.868,5.526,148.930
C02382=1207.344,-16.439,-42.006,-179.865,5.526,148.929
C02383=1207.339,-16.189,-42.019,-179.863,5.526,148.929
C02384=1207.334,-15.939,-42.032,-179.861,5.527,148.928
C02385=1207.329,-15.690,-42.046,-179.859,5.527,148.927
C02386=1207.324,-15.440,-42.059,-179.856,5.528,148.927
C02387=1207.318,-15.191,-42.073,-179.853,5.528,148.926
C02388=1207.314,-14.941,-42.086,-179.851,5.528,148.925
C02389=1207.309,-14.692,-42.100,-179.848,5.529,148.925
C02390=1207.303,-14.442,-42.113,-179.846,5.529,148.924
C02391=1207.299,-14.192,-42.126,-179.843,5.529,148.923
C02392=1207.293,-13.943,-42.140,-179.841,5.530,148.923
C02393=1207.288,-13.693,-42.153,-179.838,5.530,148.922
C02394=1207.283,-13.444,-42.167,-179.836,5.530,148.921
C02395=1207.278,-13.194,-42.181,-179.834,5.531,148.921
C02396=1207.273,-12.945,-42.194,-179.831,5.531,148.920
C02397=1207.268,-12.695,-42.208,-179.828,5.532,148.919
C02398=1207.263,-12.446,-42.221,-179.826,5.532,148.919
C02399=1207.258,-12.196,-42.235,-179.824,5.532,148.918
C02400=1207.253,-11.946,-42.249,-179.821,5.532,148.917
C02401=1207.248,-11.697,-42.262,-179.818,5.533,148.917
C02402=1207.242,-11.447,-42.276,-179.816,5.534,148.916
C02403=1207.238,-11.198,-42.289,-179.813,5.534,148.915
C02404=1207.232,-10.948,-42.303,-179.811,5.534,148.915
C02405=1207.227,-10.699,-42.316,-179.809,5.534,148.914
C02406=1207.222,-10.449,-42.329,-179.806,5.535,148.913
C02407=1207.217,-10.199,-42.344,-179.803,5.535,148.913
C02408=1207.212,-9.950,-42.358,-179.801,5.536,148.912
C02409=1207.207,-9.700,-42.371,-179.799,5.535,148.911
C02410=1207.202,-9.451,-42.385,-179.796,5.536,148.911
C02411=1207.196,-9.201,-42.398,-179.794,5.537,148.910
C02412=1207.192,-8.951,-42.412,-179.791,5.537,148.909
C02413=1207.187,-8.702,-42.426,-179.789,5.538,148.909
C02414=1207.181,-8.452,-42.439,-179.786,5.537,148.908
C02415=1207.176,-8.202,-42.454,-179.784,5.538,148.907
C02416=1207.172,-7.954,-42.467,-179.781,5.538,148.907
C02417=1207.166,-7.703,-42.480,-179.778,5.539,148.906
C02418=1207.161,-7.454,-42.494,-179.776,5.540,148.906
C02419=1207.157,-7.205,-42.508,-179.774,5.540,148.905
C02420=1207.151,-6.954,-42.522,-179.772,5.540,148.904
C02421=1207.146,-6.705,-42.535,-179.769,5.541,148.903
C02422=1207.141,-6.456,-42.550,-179.766,5.541,148.903
C02423=1207.136,-6.206,-42.563,-179.764,5.541,148.902
C02424=1207.131,-5.957,-42.577,-179.762,5.541,148.901
C02425=1207.126,-5.707,-42.591,-179.759,5.542,148.901
C02426=1207.121,-5.457,-42.605,-179.756,5.542,148.900
C02427=1207.116,-5.208,-42.618,-179.754,5.543,148.900
C02428=1207.111,-4.958,-42.632,-179.751,5.544,148.899
C02429=1207.106,-4.709,-42.646,-179.749,5.544,148.898
C02430=1207.100,-4.460,-42.660,-179.747,5.544,148.897
C02431=1207.095,-4.209,-42.674,-179.744,5.544,148.897
C02432=1207.091,-3.960,-42.687,-179.741,5.545,148.896
C02433=1207.085,-3.711,-42.701,-179.739,5.545,148.895
C02434=1207.080,-3.461,-42.716,-179.736,5.546,148.895
C02435=1207.075,-3.211,-42.730,-179.734,5.546,148.894
C02436=1207.069,-2.962,-42.743,-179.732,5.546,148.894
C02437=1207.065,-2.712,-42.757,-179.729,5.547,148.893
C02438=1207.060,-2.463,-42.771,-179.727,5.547,148.892
C02439=1207.055,-2.213,-42.785,-179.724,5.548,148.892
C02440=1207.050,-1.964,-42.799,-179.721,5.548,148.891
C02441=1207.045,-1.714,-42.814,-179.719,5.548,148.890
C02442=1207.040,-1.464,-42.827,-179.717,5.549,148.890
C02443=1207.034,-1.215,-42.841,-179.714,5.549,148.889
C02444=1207.029,-0.965,-42.855,-179.712,5.550,148.888
C02445=1207.025,-0.716,-42.869,-179.709,5.550,148.888
C02446=1207.020,-0.466,-42.883,-179.706,5.551,148.887
C02447=1207.014,-0.217,-42.897,-179.704,5.550,148.886
C02448=1207.009,0.033,-42.911,-179.702,5.551,148.886
C02449=1207.004,0.282,-42.926,-179.699,5.551,148.885
C02450=1206.999,0.532,-42.940,-179.697,5.552,148.884
C02451=1206.994,0.782,-42.953,-179.694,5.553,148.884
C02452=1206.989,1.031,-42.967,-179.691,5.553,148.883
C02453=1206.984,1.281,-42.982,-179.689,5.553,148.882
C02454=1206.979,1.531,-42.996,-179.687,5.554,148.882
C02455=1206.973,1.780,-43.010,-179.684,5.554,148.881
C02456=1206.969,2.029,-43.024,-179.681,5.555,148.880
C02457=1206.964,2.279,-43.038,-179.679,5.555,148.880
C02458=1206.959,2.529,-43.052,-179.677,5.556,148.879
C02459=1206.953,2.797,-43.068,-179.674,5.556,148.878
C02460=1206.947,3.066,-43.083,-179.671,5.557,148.878
C02461=1206.942,3.335,-43.099,-179.668,5.557,148.877
C02462=1206.937,3.605,-43.114,-179.666,5.558,148.876
C02463=1206.932,3.854,-43.128,-179.663,5.558,148.875
C02464=1206.927,4.104,-43.142,-179.661,5.558,148.875
C02465=1206.921,4.353,-43.156,-179.659,5.559,148.874
C02466=1206.916,4.603,-43.171,-179.656,5.559,148.874
C02467=1206.911,4.853,-43.185,-179.653,5.560,148.873
C02468=1206.906,5.102,-43.199,-179.651,5.560,148.872
C02469=1206.901,5.352,-43.213,-179.648,5.561,148.872
C02470=1206.896,5.602,-43.228,-179.645,5.561,148.871
C02471=1206.891,5.850,-43.242,-179.643,5.561,148.870
C02472=1206.886,6.100,-43.257,-179.641,5.562,148.870
C02473=1206.881,6.349,-43.271,-179.639,5.562,148.869
C02474=1206.876,6.599,-43.285,-179.636,5.563,148.868
C02475=1206.871,6.849,-43.299,-179.633,5.563,148.868
C02476=1206.866,7.099,-43.314,-179.631,5.564,148.867
C02477=1206.861,7.348,-43.328,-179.628,5.564,148.866
C02478=1206.856,7.597,-43.342,-179.625,5.565,148.866
C02479=1206.851,7.846,-43.357,-179.624,5.565,148.865
C02480=1206.846,8.096,-43.371,-179.621,5.565,148.864
C02481=1206.841,8.346,-43.385,-179.618,5.566,148.864
C02482=1206.836,8.596,-43.400,-179.616,5.566,148.863
C02483=1206.831,8.845,-43.414,-179.613,5.567,148.862
C02484=1206.825,9.095,-43.428,-179.610,5.567,148.862
C02485=1206.820,9.344,-43.443,-179.608,5.568,148.861
C02486=1206.815,9.593,-43.458,-179.606,5.569,148.861
C02487=1206.811,9.843,-43.472,-179.604,5.568,148.860
C02488=1206.806,10.093,-43.486,-179.601,5.569,148.859
C02489=1206.801,10.342,-43.501,-179.598,5.569,148.859
C02490=1206.796,10.592,-43.516,-179.596,5.570,148.858
C02491=1206.791,10.841,-43.530,-179.593,5.570,148.857
C02492=1206.785,11.091,-43.545,-179.590,5.571,148.856
C02493=1206.781,11.340,-43.560,-179.588,5.572,148.856
C02494=1206.775,11.589,-43.574,-179.585,5.572,148.855
C02495=1206.770,11.839,-43.588,-179.583,5.573,148.855
C02496=1206.766,12.088,-43.603,-179.581,5.573,148.854
C02497=1206.761,12.338,-43.617,-179.578,5.573,148.853
C02498=1206.755,12.588,-43.632,-179.575,5.574,148.853
C02499=1206.750,12.838,-43.646,-179.573,5.574,148.852
C02500=1206.745,13.087,-43.661,-179.571,5.575,148.851
C02501=1206.740,13.336,-43.676,-179.568,5.576,148.851
C02502=1206.735,13.586,-43.690,-179.565,5.576,148.850
C02503=1206.730,13.836,-43.705,-179.563,5.577,148.849
C02504=1206.725,14.085,-43.720,-179.560,5.577,148.849
C02505=1206.720,14.334,-43.735,-179.558,5.577,148.848
C02506=1206.715,14.584,-43.749,-179.556,5.578,148.848
C02507=1206.710,14.834,-43.763,-179.553,5.578,148.847
C02508=1206.705,15.083,-43.779,-179.551,5.579,148.846
C02509=1206.700,15.333,-43.793,-179.548,5.579,148.846
C02510=1206.695,15.583,-43.807,-179.545,5.580,148.845
C02511=1206.691,15.832,-43.822,-179.543,5.580,148.844
C02512=1206.685,16.082,-43.837,-179.540,5.581,148.844
C02513=1206.680,16.331,-43.852,-179.538,5.582,148.843
C02514=1206.675,16.581,-43.867,-179.535,5.582,148.842
C02515=1206.670,16.829,-43.881,-179.532,5.583,148.842
C02516=1206.664,17.079,-43.896,-179.530,5.582,148.841
C02517=1206.660,17.328,-43.911,-179.528,5.583,148.840
C02518=1206.655,17.578,-43.925,-179.525,5.583,148.840
C02519=1206.650,17.828,-43.941,-179.523,5.584,148.839
C02520=1206.645,18.078,-43.956,-179.520,5.585,148.838
C02521=1206.640,18.327,-43.971,-179.518,5.585,148.838
C02522=1206.635,18.577,-43.985,-179.515,5.586,148.837
C02523=1206.630,18.826,-44.000,-179.512,5.586,148.836
C02524=1206.625,19.076,-44.015,-179.510,5.587,148.836
C02525=1206.620,19.325,-44.030,-179.508,5.588,148.835
C02526=1206.615,19.575,-44.045,-179.505,5.588,148.835
C02527=1206.610,19.824,-44.060,-179.502,5.589,148.834
C02528=1206.604,20.074,-44.074,-179.500,5.589,148.833
C02529=1206.600,20.323,-44.089,-179.498,5.589,148.833
C02530=1206.595,20.573,-44.104,-179.495,5.589,148.832
C02531=1206.589,20.822,-44.119,-179.493,5.590,148.831
C02532=1206.585,21.071,-44.134,-179.490,5.591,148.831
C02533=1206.580,21.321,-44.149,-179.487,5.591,148.830
C02534=1206.574,21.570,-44.164,-179.485,5.592,148.829
C02535=1206.569,21.820,-44.178,-179.482,5.592,148.829
C02536=1206.564,22.069,-44.194,-179.479,5.593,148.828
C02537=1206.559,22.318,-44.209,-179.477,5.594,148.828
C02538=1206.554,22.568,-44.223,-179.475,5.594,148.827
C02539=1206.549,22.817,-44.239,-179.472,5.595,148.826
C02540=1206.545,23.067,-44.254,-179.469,5.595,148.826
C02541=1206.539,23.317,-44.269,-179.467,5.596,148.825
C02542=1206.535,23.566,-44.284,-179.464,5.596,148.824
C02543=1206.529,23.816,-44.300,-179.462,5.597,148.824
C02544=1206.524,24.065,-44.314,-179.459,5.598,148.823
C02545=1206.520,24.315,-44.329,-179.457,5.598,148.822
C02546=1206.514,24.564,-44.345,-179.455,5.598,148.822
C02547=1206.509,24.814,-44.359,-179.452,5.599,148.821
C02548=1206.504,25.063,-44.374,-179.450,5.599,148.821
C02549=1206.500,25.313,-44.390,-179.447,5.600,148.820
C02550=1206.494,25.562,-44.405,-179.444,5.600,148.819
C02551=1206.489,25.812,-44.420,-179.442,5.601,148.819
C02552=1206.484,26.061,-44.435,-179.439,5.602,148.818
C02553=1206.479,26.310,-44.450,-179.437,5.602,148.817
C02554=1206.474,26.560,-44.466,-179.434,5.603,148.817
C02555=1206.469,26.810,-44.480,-179.432,5.603,148.816
C02556=1206.464,27.059,-44.496,-179.429,5.604,148.815
C02557=1206.460,27.309,-44.511,-179.426,5.605,148.815
C02558=1206.454,27.558,-44.527,-179.424,5.605,148.814
C02559=1206.450,27.807,-44.542,-179.421,5.606,148.813
C02560=1206.444,28.057,-44.556,-179.419,5.606,148.813
C02561=1206.439,28.306,-44.571,-179.416,5.607,148.812
C02562=1206.434,28.556,-44.587,-179.414,5.607,148.812
C02563=1206.429,28.825,-44.604,-179.411,5.608,148.811
C02564=1206.424,29.094,-44.620,-179.408,5.609,148.810
C02565=1206.418,29.362,-44.637,-179.406,5.609,148.809
C02566=1206.413,29.631,-44.653,-179.403,5.610,148.809
C02567=1206.408,29.880,-44.668,-179.401,5.610,148.808
C02568=1206.402,30.130,-44.684,-179.398,5.611,148.807
C02569=1206.398,30.379,-44.699,-179.395,5.611,148.807
C02570=1206.393,30.629,-44.715,-179.393,5.612,148.806
C02571=1206.388,30.878,-44.730,-179.390,5.613,148.806
C02572=1206.383,31.128,-44.746,-179.388,5.613,148.805
C02573=1206.378,31.377,-44.761,-179.385,5.614,148.804
C02574=1206.373,31.627,-44.775,-179.382,5.614,148.804
C02575=1206.368,31.877,-44.791,-179.380,5.615,148.803
C02576=1206.362,32.126,-44.807,-179.378,5.616,148.802
C02577=1206.358,32.375,-44.822,-179.375,5.616,148.802
C02578=1206.352,32.625,-44.838,-179.372,5.617,148.801
C02579=1206.348,32.874,-44.853,-179.370,5.617,148.800
C02580=1206.343,33.124,-44.868,-179.368,5.618,148.800
C02581=1206.338,33.373,-44.884,-179.365,5.619,148.799
C02582=1206.333,33.622,-44.899,-179.362,5.619,148.799
C02583=1206.328,33.872,-44.915,-179.360,5.620,148.798
C02584=1206.323,34.122,-44.931,-179.357,5.620,148.797
C02585=1206.318,34.371,-44.946,-179.355,5.621,148.797
C02586=1206.313,34.620,-44.961,-179.352,5.622,148.796
C02587=1206.308,34.870,-44.977,-179.350,5.622,148.796
C02588=1206.303,35.119,-44.993,-179.347,5.623,148.795
C02589=1206.298,35.368,-45.008,-179.344,5.623,148.794
C02590=1206.293,35.618,-45.024,-179.342,5.624,148.794
C02591=1206.288,35.868,-45.040,-179.340,5.625,148.793
C02592=1206.283,36.117,-45.055,-179.337,5.625,148.792
C02593=1206.278,36.366,-45.071,-179.334,5.626,148.792
C02594=1206.273,36.616,-45.087,-179.332,5.626,148.791
C02595=1206.268,36.866,-45.102,-179.329,5.627,148.791
C02596=1206.263,37.115,-45.117,-179.327,5.628,148.790
C02597=1206.258,37.364,-45.133,-179.324,5.628,148.789
C02598=1206.253,37.614,-45.149,-179.322,5.629,148.789
C02599=1206.248,37.863,-45.165,-179.319,5.629,148.788
C02600=1206.242,38.113,-45.181,-179.317,5.630,148.787
C02601=1206.238,38.362,-45.196,-179.314,5.631,148.787
C02602=1206.233,38.612,-45.211,-179.311,5.631,148.786
C02603=1206.228,38.861,-45.227,-179.309,5.632,148.785
C02604=1206.223,39.111,-45.244,-179.307,5.633,148.785
C02605=1206.218,39.360,-45.259,-179.304,5.633,148.784
C02606=1206.213,39.609,-45.274,-179.301,5.634,148.784
C02607=1206.208,39.859,-45.290,-179.299,5.634,148.783
C02608=1206.203,40.109,-45.306,-179.296,5.635,148.782
C02609=1206.198,40.357,-45.322,-179.294,5.636,148.782
C02610=1206.193,40.608,-45.338,-179.291,5.636,148.781
C02611=1206.188,40.857,-45.353,-179.289,5.637,148.780
C02612=1206.184,41.107,-45.369,-179.286,5.637,148.780
C02613=1206.179,41.356,-45.385,-179.284,5.638,148.779
C02614=1206.173,41.605,-45.401,-179.281,5.639,148.779
C02615=1206.168,41.855,-45.417,-179.278,5.640,148.778
C02616=1206.163,42.104,-45.433,-179.275,5.641,148.777
C02617=1206.158,42.353,-45.449,-179.273,5.641,148.777
C02618=1206.153,42.603,-45.465,-179.271,5.642,148.776
C02619=1206.149,42.852,-45.480,-179.268,5.643,148.776
C02620=1206.144,43.102,-45.496,-179.265,5.643,148.775
C02621=1206.139,43.351,-45.512,-179.263,5.644,148.774
C02622=1206.133,43.601,-45.528,-179.260,5.644,148.774
C02623=1206.129,43.850,-45.544,-179.258,5.645,148.773
C02624=1206.123,44.100,-45.560,-179.255,5.646,148.772
C02625=1206.119,44.349,-45.577,-179.253,5.646,148.772
C02626=1206.114,44.598,-45.592,-179.250,5.647,148.771
C02627=1206.108,44.848,-45.608,-179.248,5.648,148.771
C02628=1206.104,45.097,-45.624,-179.245,5.648,148.770
C02629=1206.098,45.347,-45.640,-179.243,5.649,148.769
C02630=1206.094,45.596,-45.657,-179.240,5.649,148.769
C02631=1206.088,45.846,-45.672,-179.238,5.650,148.768
C02632=1206.084,46.096,-45.688,-179.235,5.651,148.767
C02633=1206.079,46.345,-45.704,-179.232,5.651,148.767
C02634=1206.074,46.594,-45.720,-179.230,5.652,148.766
C02635=1206.069,46.843,-45.736,-179.228,5.653,148.766
C02636=1206.064,47.093,-45.752,-179.224,5.654,148.765
C02637=1206.060,47.342,-45.768,-179.222,5.654,148.764
C02638=1206.054,47.591,-45.784,-179.219,5.655,148.764
C02639=1206.050,47.841,-45.801,-179.217,5.656,148.763
C02640=1206.044,48.090,-45.816,-179.214,5.656,148.763
C02641=1206.040,48.340,-45.833,-179.212,5.657,148.762
C02642=1206.034,48.590,-45.849,-179.209,5.658,148.761
C02643=1206.029,48.839,-45.866,-179.206,5.658,148.761
C02644=1206.024,49.088,-45.881,-179.204,5.659,148.760
C02645=1206.019,49.338,-45.898,-179.202,5.660,148.759
C02646=1206.014,49.587,-45.914,-179.199,5.660,148.759
C02647=1206.009,49.837,-45.930,-179.196,5.661,148.758
C02648=1206.004,50.086,-45.947,-179.194,5.661,148.758
C02649=1206.000,50.336,-45.963,-179.192,5.662,148.757
C02650=1205.995,50.584,-45.979,-179.188,5.663,148.756
C02651=1205.990,50.835,-45.995,-179.186,5.664,148.756
C02652=1205.985,51.083,-46.011,-179.184,5.665,148.755
C02653=1205.980,51.333,-46.027,-179.181,5.665,148.755
C02654=1205.975,51.582,-46.043,-179.178,5.666,148.754
C02655=1205.970,51.832,-46.060,-179.176,5.666,148.753
C02656=1205.966,52.082,-46.076,-179.174,5.667,148.753
C02657=1205.960,52.331,-46.093,-179.171,5.668,148.752
C02658=1205.955,52.580,-46.110,-179.168,5.668,148.751
C02659=1205.950,52.830,-46.125,-179.166,5.669,148.751
C02660=1205.945,53.079,-46.142,-179.164,5.670,148.750
C02661=1205.940,53.328,-46.158,-179.161,5.670,148.750
C02662=1205.935,53.578,-46.174,-179.158,5.672,148.749
C02663=1205.930,53.827,-46.190,-179.156,5.673,148.749
C02664=1205.925,54.077,-46.208,-179.153,5.673,148.748
C02665=1205.921,54.326,-46.224,-179.150,5.674,148.747
C02666=1205.915,54.576,-46.240,-179.148,5.674,148.747
C02667=1205.911,54.844,-46.258,-179.145,5.675,148.746
C02668=1205.905,55.113,-46.275,-179.142,5.675,148.745
C02669=1205.899,55.381,-46.293,-179.139,5.677,148.745
C02670=1205.894,55.649,-46.311,-179.137,5.678,148.744
C02671=1205.889,55.899,-46.327,-179.134,5.678,148.743
C02672=1205.885,56.148,-46.344,-179.132,5.679,148.743
C02673=1205.879,56.398,-46.361,-179.129,5.679,148.742
C02674=1205.874,56.647,-46.377,-179.127,5.680,148.742
C02675=1205.870,56.897,-46.393,-179.124,5.682,148.741
C02676=1205.864,57.146,-46.409,-179.121,5.682,148.740
C02677=1205.860,57.395,-46.426,-179.118,5.683,148.740
C02678=1205.855,57.645,-46.443,-179.116,5.684,148.739
C02679=1205.850,57.894,-46.460,-179.114,5.684,148.739
C02680=1205.845,58.143,-46.476,-179.111,5.685,148.738
C02681=1205.840,58.393,-46.492,-179.109,5.686,148.738
C02682=1205.835,58.642,-46.509,-179.106,5.686,148.737
C02683=1205.830,58.892,-46.526,-179.104,5.687,148.736
C02684=1205.825,59.141,-46.542,-179.100,5.688,148.736
C02685=1205.820,59.391,-46.559,-179.098,5.689,148.735
C02686=1205.815,59.640,-46.576,-179.096,5.690,148.734
C02687=1205.810,59.889,-46.592,-179.093,5.690,148.734
C02688=1205.805,60.139,-46.610,-179.091,5.691,148.733
C02689=1205.801,60.388,-46.626,-179.088,5.692,148.733
C02690=1205.795,60.637,-46.643,-179.086,5.692,148.732
C02691=1205.791,60.886,-46.659,-179.082,5.693,148.731
C02692=1205.786,61.136,-46.677,-179.080,5.694,148.731
C02693=1205.780,61.386,-46.692,-179.078,5.695,148.730
C02694=1205.776,61.635,-46.709,-179.075,5.695,148.730
C02695=1205.771,61.885,-46.726,-179.073,5.696,148.729
C02696=1205.766,62.134,-46.743,-179.070,5.697,148.728
C02697=1205.760,62.383,-46.760,-179.068,5.698,148.728
C02698=1205.756,62.633,-46.776,-179.065,5.698,148.727
C02699=1205.751,62.882,-46.793,-179.062,5.700,148.727
C02700=1205.746,63.131,-46.810,-179.060,5.700,148.726
C02701=1205.741,63.380,-46.827,-179.057,5.701,148.725
C02702=1205.737,63.630,-46.844,-179.055,5.702,148.725
C02703=1205.732,63.880,-46.861,-179.052,5.702,148.724
C02704=1205.727,64.128,-46.878,-179.050,5.703,148.724
C02705=1205.721,64.378,-46.895,-179.046,5.704,148.723
C02706=1205.717,64.628,-46.912,-179.044,5.705,148.723
C02707=1205.712,64.876,-46.928,-179.042,5.706,148.722
C02708=1205.707,65.126,-46.945,-179.039,5.706,148.721
C02709=1205.702,65.376,-46.962,-179.037,5.707,148.721
C02710=1205.697,65.626,-46.979,-179.034,5.708,148.720
C02711=1205.692,65.875,-46.996,-179.032,5.708,148.719
C02712=1205.687,66.124,-47.013,-179.029,5.710,148.719
C02713=1205.682,66.373,-47.030,-179.026,5.711,148.718
C02714=1205.677,66.623,-47.047,-179.024,5.711,148.718
C02715=1205.673,66.872,-47.064,-179.021,5.712,148.717
C02716=1205.667,67.121,-47.081,-179.019,5.713,148.717
C02717=1205.662,67.371,-47.097,-179.016,5.713,148.716
C02718=1205.657,67.621,-47.115,-179.013,5.715,148.715
C02719=1205.653,67.869,-47.132,-179.011,5.715,148.715
C02720=1205.648,68.119,-47.149,-179.008,5.716,148.714
C02721=1205.643,68.368,-47.166,-179.006,5.717,148.714
C02722=1205.638,68.618,-47.183,-179.003,5.718,148.713
C02723=1205.633,68.867,-47.200,-179.001,5.718,148.712
C02724=1205.628,69.117,-47.218,-178.998,5.719,148.712
C02725=1205.624,69.366,-47.234,-178.995,5.720,148.711
C02726=1205.618,69.615,-47.251,-178.993,5.721,148.711
C02727=1205.614,69.864,-47.269,-178.990,5.721,148.710
C02728=1205.608,70.114,-47.286,-178.988,5.722,148.710
C02729=1205.604,70.363,-47.302,-178.985,5.724,148.709
C02730=1205.599,70.613,-47.320,-178.982,5.724,148.708
C02731=1205.595,70.862,-47.337,-178.980,5.725,148.708
C02732=1205.589,71.111,-47.354,-178.977,5.726,148.707
C02733=1205.584,71.361,-47.371,-178.975,5.726,148.707
C02734=1205.579,71.610,-47.389,-178.972,5.728,148.706
C02735=1205.574,71.859,-47.406,-178.969,5.729,148.705
C02736=1205.570,72.109,-47.423,-178.967,5.729,148.705
C02737=1205.565,72.358,-47.441,-178.965,5.730,148.704
C02738=1205.560,72.608,-47.458,-178.962,5.731,148.704
C02739=1205.554,72.857,-47.474,-178.959,5.731,148.703
C02740=1205.550,73.106,-47.492,-178.957,5.733,148.703
C02741=1205.544,73.356,-47.509,-178.954,5.734,148.702
C02742=1205.540,73.605,-47.527,-178.951,5.734,148.701
C02743=1205.535,73.854,-47.544,-178.949,5.735,148.701
C02744=1205.530,74.104,-47.561,-178.947,5.736,148.700
C02745=1205.526,74.353,-47.579,-178.943,5.737,148.700
C02746=1205.520,74.603,-47.596,-178.941,5.738,148.699
C02747=1205.516,74.852,-47.613,-178.939,5.738,148.698
C02748=1205.510,75.101,-47.630,-178.936,5.739,148.698
C02749=1205.505,75.350,-47.648,-178.933,5.741,148.697
C02750=1205.501,75.599,-47.665,-178.931,5.741,148.697
C02751=1205.496,75.849,-47.683,-178.928,5.742,148.696
C02752=1205.491,76.098,-47.700,-178.926,5.743,148.696
C02753=1205.486,76.348,-47.718,-178.923,5.743,148.695
C02754=1205.481,76.597,-47.735,-178.920,5.745,148.694
C02755=1205.477,76.846,-47.753,-178.918,5.746,148.694
C02756=1205.471,77.096,-47.770,-178.915,5.746,148.693
C02757=1205.467,77.345,-47.787,-178.913,5.747,148.693
C02758=1205.462,77.595,-47.805,-178.910,5.749,148.692
C02759=1205.457,77.844,-47.823,-178.907,5.749,148.691
C02760=1205.452,78.094,-47.840,-178.905,5.750,148.691
C02761=1205.448,78.342,-47.857,-178.903,5.751,148.690
C02762=1205.443,78.592,-47.875,-178.900,5.751,148.690
C02763=1205.437,78.841,-47.893,-178.897,5.753,148.689
C02764=1205.433,79.091,-47.911,-178.895,5.753,148.689
C02765=1205.427,79.340,-47.927,-178.892,5.754,148.688
C02766=1205.423,79.589,-47.945,-178.890,5.755,148.688
C02767=1205.418,79.838,-47.963,-178.887,5.756,148.687
C02768=1205.412,80.088,-47.980,-178.884,5.757,148.686
C02769=1205.408,80.337,-47.998,-178.882,5.758,148.686
C02770=1205.403,80.586,-48.016,-178.879,5.758,148.685
C02771=1205.397,80.855,-48.035,-178.876,5.760,148.685
C02772=1205.393,81.123,-48.054,-178.873,5.760,148.684
C02773=1205.388,81.392,-48.072,-178.871,5.762,148.683
C02774=1205.382,81.660,-48.092,-178.868,5.763,148.683
C02775=1205.378,81.909,-48.110,-178.866,5.763,148.682
C02776=1205.372,82.159,-48.127,-178.863,5.764,148.682
C02777=1205.367,82.408,-48.145,-178.860,5.766,148.681
C02778=1205.362,82.657,-48.163,-178.858,5.766,148.680
C02779=1205.357,82.907,-48.180,-178.855,5.767,148.680
C02780=1205.352,83.156,-48.198,-178.853,5.768,148.679
C02781=1205.348,83.405,-48.215,-178.850,5.769,148.679
C02782=1205.343,83.654,-48.233,-178.847,5.770,148.678
C02783=1205.338,83.904,-48.251,-178.845,5.770,148.678
C02784=1205.333,84.153,-48.269,-178.842,5.772,148.677
C02785=1205.328,84.402,-48.287,-178.840,5.773,148.677
C02786=1205.323,84.652,-48.305,-178.837,5.773,148.676
C02787=1205.318,84.901,-48.323,-178.835,5.774,148.675
C02788=1205.313,85.150,-48.341,-178.832,5.776,148.675
C02789=1205.308,85.400,-48.358,-178.829,5.776,148.674
C02790=1205.304,85.650,-48.376,-178.827,5.777,148.674
C02791=1205.299,85.899,-48.394,-178.824,5.778,148.673
C02792=1205.294,86.148,-48.412,-178.821,5.779,148.673
C02793=1205.289,86.397,-48.430,-178.819,5.780,148.672
C02794=1205.284,86.646,-48.448,-178.816,5.781,148.671
C02795=1205.279,86.895,-48.466,-178.814,5.782,148.671
C02796=1205.274,87.145,-48.483,-178.811,5.783,148.670
C02797=1205.270,87.394,-48.501,-178.809,5.784,148.670
C02798=1205.265,87.643,-48.519,-178.806,5.784,148.669
C02799=1205.260,87.892,-48.537,-178.803,5.786,148.669
C02800=1205.255,88.143,-48.556,-178.801,5.787,148.668
C02801=1205.250,88.392,-48.574,-178.798,5.787,148.668
C02802=1205.245,88.641,-48.592,-178.796,5.788,148.667
C02803=1205.240,88.890,-48.610,-178.793,5.790,148.666
C02804=1205.235,89.139,-48.628,-178.790,5.790,148.666
C02805=1205.231,89.388,-48.646,-178.788,5.791,148.665
C02806=1205.226,89.638,-48.664,-178.785,5.793,148.665
C02807=1205.221,89.888,-48.682,-178.783,5.793,148.664
C02808=1205.216,90.137,-48.700,-178.780,5.794,148.664
C02809=1205.212,90.386,-48.718,-178.777,5.796,148.663
C02810=1205.207,90.635,-48.736,-178.775,5.796,148.663
C02811=1205.202,90.884,-48.754,-178.772,5.797,148.662
C02812=1205.197,91.133,-48.772,-178.770,5.798,148.662
C02813=1205.192,91.383,-48.790,-178.767,5.799,148.661
C02814=1205.188,91.632,-48.808,-178.765,5.800,148.660
C02815=1205.183,91.882,-48.826,-178.762,5.801,148.660
C02816=1205.177,92.131,-48.845,-178.759,5.802,148.659
C02817=1205.172,92.380,-48.863,-178.757,5.803,148.659
C02818=1205.167,92.629,-48.881,-178.754,5.804,148.658
C02819=1205.163,92.879,-48.900,-178.751,5.805,148.658
C02820=1205.158,93.128,-48.918,-178.749,5.806,148.657
C02821=1205.153,93.377,-48.936,-178.747,5.807,148.657
C02822=1205.148,93.626,-48.954,-178.744,5.808,148.656
C02823=1205.144,93.875,-48.972,-178.741,5.809,148.655
C02824=1205.138,94.126,-48.991,-178.739,5.810,148.655
C02825=1205.134,94.375,-49.009,-178.736,5.810,148.654
C02826=1205.129,94.623,-49.027,-178.733,5.812,148.654
C02827=1205.124,94.873,-49.045,-178.731,5.813,148.653
C02828=1205.120,95.122,-49.064,-178.729,5.814,148.653
C02829=1205.114,95.372,-49.082,-178.726,5.815,148.652
C02830=1205.109,95.621,-49.100,-178.723,5.816,148.651
C02831=1205.105,95.870,-49.119,-178.721,5.817,148.651
C02832=1205.100,96.120,-49.137,-178.718,5.818,148.650
C02833=1205.095,96.369,-49.155,-178.715,5.819,148.650
C02834=1205.090,96.618,-49.174,-178.713,5.819,148.649
C02835=1205.085,96.867,-49.192,-178.710,5.821,148.649
C02836=1205.081,97.117,-49.211,-178.708,5.822,148.648
C02837=1205.076,97.366,-49.229,-178.705,5.822,148.648
C02838=1205.070,97.615,-49.247,-178.702,5.824,148.647
C02839=1205.066,97.864,-49.266,-178.700,5.825,148.647
C02840=1205.061,98.114,-49.284,-178.697,5.826,148.646
C02841=1205.056,98.363,-49.302,-178.694,5.827,148.646
C02842=1205.051,98.612,-49.322,-178.692,5.828,148.645
C02843=1205.047,98.862,-49.340,-178.689,5.829,148.644
C02844=1205.042,99.111,-49.358,-178.687,5.830,148.644
C02845=1205.036,99.360,-49.377,-178.684,5.831,148.643
C02846=1205.032,99.610,-49.396,-178.681,5.833,148.643
C02847=1205.027,99.859,-49.414,-178.679,5.833,148.642
C02848=1205.023,100.107,-49.432,-178.676,5.834,148.642
C02849=1205.018,100.357,-49.451,-178.674,5.836,148.641
C02850=1205.013,100.607,-49.469,-178.671,5.836,148.641
C02851=1205.008,100.855,-49.488,-178.669,5.837,148.640
C02852=1205.003,101.105,-49.507,-178.666,5.839,148.640
C02853=1204.998,101.354,-49.526,-178.663,5.839,148.639
C02854=1204.994,101.603,-49.543,-178.661,5.840,148.639
C02855=1204.989,101.853,-49.563,-178.658,5.842,148.638
C02856=1204.984,102.102,-49.581,-178.656,5.842,148.637
C02857=1204.979,102.351,-49.600,-178.653,5.844,148.637
C02858=1204.974,102.601,-49.619,-178.650,5.845,148.636
C02859=1204.969,102.850,-49.637,-178.648,5.846,148.636
C02860=1204.964,103.099,-49.656,-178.645,5.847,148.635
C02861=1204.960,103.349,-49.674,-178.643,5.848,148.635
C02862=1204.954,103.597,-49.694,-178.640,5.849,148.634
C02863=1204.949,103.847,-49.712,-178.637,5.850,148.634
C02864=1204.945,104.096,-49.731,-178.635,5.851,148.633
C02865=1204.940,104.345,-49.750,-178.632,5.852,148.633
C02866=1204.936,104.595,-49.768,-178.630,5.853,148.632
C02867=1204.930,104.843,-49.788,-178.627,5.854,148.632
C02868=1204.925,105.093,-49.806,-178.624,5.856,148.631
C02869=1204.921,105.342,-49.825,-178.622,5.856,148.631
C02870=1204.916,105.591,-49.843,-178.619,5.857,148.630
C02871=1204.911,105.841,-49.863,-178.616,5.859,148.629
C02872=1204.906,106.089,-49.882,-178.614,5.859,148.629
C02873=1204.902,106.339,-49.900,-178.611,5.861,148.628
C02874=1204.897,106.588,-49.919,-178.609,5.862,148.628
C02875=1204.891,106.857,-49.939,-178.606,5.863,148.627
C02876=1204.887,107.125,-49.960,-178.603,5.864,148.627
C02877=1204.881,107.394,-49.980,-178.600,5.866,148.626
C02878=1204.876,107.662,-50.001,-178.598,5.866,148.626
C02879=1204.871,107.911,-50.020,-178.595,5.868,148.625
C02880=1204.866,108.160,-50.038,-178.592,5.869,148.625
C02881=1204.862,108.410,-50.057,-178.590,5.870,148.624
C02882=1204.856,108.659,-50.076,-178.587,5.871,148.624
C02883=1204.852,108.908,-50.095,-178.585,5.872,148.623
C02884=1204.847,109.157,-50.114,-178.582,5.873,148.623
C02885=1204.842,109.407,-50.134,-178.580,5.874,148.622
C02886=1204.837,109.655,-50.152,-178.576,5.876,148.622
C02887=1204.832,109.906,-50.171,-178.574,5.877,148.621
C02888=1204.828,110.154,-50.190,-178.572,5.877,148.620
C02889=1204.823,110.404,-50.210,-178.569,5.879,148.620
C02890=1204.818,110.652,-50.228,-178.566,5.879,148.619
C02891=1204.813,110.902,-50.247,-178.564,5.881,148.619
C02892=1204.808,111.151,-50.267,-178.561,5.882,148.618
C02893=1204.804,111.401,-50.286,-178.559,5.883,148.618
C02894=1204.799,111.649,-50.305,-178.556,5.884,148.617
C02895=1204.794,111.899,-50.325,-178.554,5.885,148.617
C02896=1204.789,112.148,-50.343,-178.551,5.887,148.616
C02897=1204.784,112.398,-50.362,-178.548,5.887,148.616
C02898=1204.780,112.646,-50.381,-178.545,5.889,148.615
C02899=1204.775,112.896,-50.401,-178.543,5.890,148.615
C02900=1204.770,113.145,-50.420,-178.540,5.890,148.614
C02901=1204.766,113.394,-50.439,-178.538,5.892,148.614
C02902=1204.761,113.644,-50.459,-178.535,5.893,148.613
C02903=1204.756,113.892,-50.478,-178.532,5.895,148.613
C02904=1204.752,114.142,-50.497,-178.530,5.895,148.612
C02905=1204.746,114.391,-50.516,-178.527,5.897,148.612
C02906=1204.741,114.641,-50.535,-178.525,5.898,148.611
C02907=1204.736,114.890,-50.555,-178.522,5.899,148.611
C02908=1204.732,115.139,-50.574,-178.520,5.900,148.610
C02909=1204.726,115.388,-50.593,-178.517,5.901,148.610
C02910=1204.722,115.637,-50.613,-178.514,5.903,148.609
C02911=1204.717,115.887,-50.632,-178.512,5.903,148.609
C02912=1204.712,116.135,-50.651,-178.509,5.905,148.608
C02913=1204.708,116.385,-50.671,-178.507,5.906,148.608
C02914=1204.702,116.634,-50.690,-178.504,5.907,148.607
C02915=1204.698,116.883,-50.709,-178.501,5.908,148.607
C02916=1204.694,117.133,-50.729,-178.499,5.910,148.606
C02917=1204.688,117.382,-50.748,-178.496,5.910,148.605
C02918=1204.683,117.631,-50.768,-178.493,5.912,148.605
C02919=1204.678,117.880,-50.787,-178.491,5.913,148.605
C02920=1204.674,118.129,-50.807,-178.488,5.914,148.604
C02921=1204.670,118.378,-50.826,-178.486,5.915,148.604
C02922=1204.664,118.627,-50.846,-178.483,5.916,148.603
C02923=1204.660,118.877,-50.865,-178.480,5.918,148.603
C02924=1204.655,119.126,-50.885,-178.478,5.918,148.602
C02925=1204.650,119.375,-50.904,-178.475,5.920,148.602
C02926=1204.645,119.624,-50.923,-178.473,5.921,148.601
C02927=1204.641,119.874,-50.943,-178.470,5.922,148.601
C02928=1204.635,120.123,-50.962,-178.468,5.923,148.600
C02929=1204.631,120.372,-50.982,-178.465,5.925,148.600
C02930=1204.626,120.621,-51.002,-178.462,5.926,148.599
C02931=1204.621,120.870,-51.021,-178.459,5.927,148.598
C02932=1204.617,121.119,-51.041,-178.457,5.928,148.598
C02933=1204.612,121.369,-51.060,-178.454,5.930,148.597
C02934=1204.607,121.618,-51.079,-178.452,5.930,148.597
C02935=1204.602,121.867,-51.100,-178.449,5.932,148.597
C02936=1204.598,122.116,-51.119,-178.447,5.933,148.596
C02937=1204.592,122.365,-51.139,-178.444,5.935,148.596
C02938=1204.587,122.615,-51.158,-178.441,5.935,148.595
C02939=1204.583,122.864,-51.179,-178.439,5.937,148.595
C02940=1204.578,123.113,-51.198,-178.436,5.938,148.594
C02941=1204.573,123.362,-51.218,-178.433,5.939,148.594
C02942=1204.568,123.612,-51.237,-178.431,5.940,148.593
C02943=1204.565,123.860,-51.257,-178.428,5.942,148.593
C02944=1204.559,124.109,-51.276,-178.426,5.943,148.592
C02945=1204.554,124.359,-51.296,-178.423,5.944,148.592
C02946=1204.550,124.608,-51.316,-178.421,5.945,148.591
C02947=1204.545,124.857,-51.336,-178.418,5.947,148.591
C02948=1204.540,125.106,-51.355,-178.415,5.947,148.590
C02949=1204.535,125.355,-51.376,-178.413,5.949,148.590
C02950=1204.531,125.605,-51.395,-178.410,5.950,148.589
C02951=1204.525,125.854,-51.415,-178.407,5.952,148.589
C02952=1204.521,126.103,-51.435,-178.405,5.953,148.588
C02953=1204.516,126.352,-51.455,-178.402,5.954,148.588
C02954=1204.512,126.601,-51.475,-178.400,5.955,148.587
C02955=1204.507,126.851,-51.495,-178.397,5.956,148.587
C02956=1204.502,127.099,-51.514,-178.395,5.957,148.586
C02957=1204.497,127.348,-51.534,-178.392,5.959,148.586
C02958=1204.493,127.598,-51.554,-178.389,5.960,148.585
C02959=1204.488,127.847,-51.575,-178.387,5.961,148.585
C02960=1204.483,128.096,-51.594,-178.384,5.962,148.584
C02961=1204.478,128.345,-51.615,-178.381,5.964,148.584
C02962=1204.473,128.595,-51.634,-178.379,5.965,148.583
C02963=1204.468,128.844,-51.655,-178.376,5.966,148.583
C02964=1204.464,129.093,-51.674,-178.374,5.967,148.582
C02965=1204.459,129.342,-51.695,-178.371,5.969,148.582
C02966=1204.454,129.591,-51.714,-178.369,5.970,148.581
C02967=1204.449,129.840,-51.734,-178.366,5.971,148.581
C02968=1204.445,130.089,-51.754,-178.363,5.972,148.580
C02969=1204.440,130.338,-51.775,-178.361,5.974,148.580
C02970=1204.435,130.588,-51.794,-178.358,5.975,148.580
C02971=1204.430,130.837,-51.815,-178.355,5.976,148.579
C02972=1204.425,131.086,-51.834,-178.353,5.978,148.578
C02973=1204.421,131.335,-51.855,-178.350,5.978,148.578
C02974=1204.416,131.584,-51.875,-178.347,5.980,148.577
C02975=1204.411,131.834,-51.895,-178.345,5.981,148.577
C02976=1204.407,132.083,-51.915,-178.342,5.983,148.576
C02977=1204.402,132.332,-51.936,-178.340,5.984,148.576
C02978=1204.396,132.581,-51.955,-178.337,5.985,148.576
C02979=1204.392,132.849,-51.978,-178.334,5.987,148.575
C02980=1204.387,133.118,-51.999,-178.332,5.987,148.574
C02981=1204.382,133.387,-52.020,-178.329,5.989,148.574
C02982=1204.376,133.655,-52.043,-178.326,5.991,148.573
C02983=1204.372,133.904,-52.063,-178.323,5.992,148.573
C02984=1204.367,134.154,-52.083,-178.321,5.993,148.573
C02985=1204.362,134.403,-52.104,-178.318,5.995,148.572
C02986=1204.358,134.652,-52.124,-178.316,5.996,148.572
C02987=1204.352,134.901,-52.143,-178.313,5.998,148.571
C02988=1204.348,135.150,-52.164,-178.310,5.998,148.571
C02989=1204.343,135.399,-52.185,-178.308,6.000,148.570
C02990=1204.338,135.648,-52.205,-178.305,6.002,148.570
C02991=1204.334,135.898,-52.225,-178.302,6.002,148.569
C02992=1204.328,136.147,-52.246,-178.300,6.004,148.569
C02993=1204.324,136.396,-52.266,-178.298,6.005,148.568
C02994=1204.320,136.645,-52.287,-178.294,6.006,148.568
C02995=1204.315,136.894,-52.307,-178.292,6.007,148.567
C02996=1204.310,137.144,-52.327,-178.290,6.009,148.567
C02997=1204.305,137.393,-52.348,-178.286,6.011,148.566
C02998=1204.301,137.642,-52.368,-178.284,6.012,148.566
C02999=1204.296,137.891,-52.389,-178.282,6.013,148.566
C03000=1204.291,138.140,-52.409,-178.279,6.014,148.565
C03001=1204.287,138.389,-52.430,-178.276,6.016,148.565
C03002=1204.281,138.638,-52.451,-178.274,6.017,148.564
C03003=1204.277,138.888,-52.470,-178.271,6.018,148.564
C03004=1204.272,139.137,-52.491,-178.268,6.020,148.563
C03005=1204.267,139.386,-52.512,-178.266,6.021,148.563
C03006=1204.263,139.635,-52.532,-178.263,6.022,148.562
C03007=1204.258,139.884,-52.552,-178.261,6.023,148.562
C03008=1204.253,140.133,-52.573,-178.258,6.025,148.561
C03009=1204.249,140.382,-52.594,-178.255,6.027,148.561
C03010=1204.243,140.631,-52.615,-178.253,6.028,148.560
C03011=1204.239,140.880,-52.635,-178.250,6.029,148.560
C03012=1204.235,141.129,-52.655,-178.248,6.030,148.559
C03013=1204.229,141.378,-52.676,-178.245,6.032,148.559
C03014=1204.225,141.627,-52.697,-178.242,6.033,148.559
C03015=1204.220,141.876,-52.718,-178.240,6.034,148.558
C03016=1204.215,142.125,-52.738,-178.237,6.036,148.558
C03017=1204.210,142.375,-52.759,-178.234,6.038,148.557
C03018=1204.206,142.624,-52.779,-178.232,6.038,148.557
C03019=1204.201,142.873,-52.800,-178.229,6.040,148.556
C03020=1204.196,143.122,-52.821,-178.227,6.041,148.556
C03021=1204.192,143.371,-52.841,-178.224,6.043,148.555
C03022=1204.187,143.620,-52.862,-178.221,6.044,148.555
C03023=1204.182,143.869,-52.882,-178.219,6.045,148.554
C03024=1204.177,144.118,-52.903,-178.216,6.047,148.554
C03025=1204.173,144.367,-52.924,-178.213,6.048,148.553
C03026=1204.168,144.616,-52.945,-178.211,6.049,148.553
C03027=1204.163,144.865,-52.966,-178.208,6.051,148.553
C03028=1204.159,145.115,-52.987,-178.206,6.052,148.552
C03029=1204.154,145.364,-53.008,-178.203,6.054,148.552
C03030=1204.149,145.613,-53.028,-178.200,6.055,148.551
C03031=1204.144,145.862,-53.049,-178.198,6.056,148.551
C03032=1204.140,146.111,-53.071,-178.195,6.058,148.550
C03033=1204.135,146.360,-53.092,-178.192,6.060,148.550
C03034=1204.130,146.609,-53.112,-178.190,6.061,148.550
C03035=1204.125,146.858,-53.133,-178.187,6.062,148.549
C03036=1204.120,147.107,-53.153,-178.185,6.064,148.549
C03037=1204.116,147.356,-53.175,-178.182,6.065,148.548
C03038=1204.111,147.606,-53.196,-178.180,6.067,148.548
C03039=1204.107,147.855,-53.217,-178.177,6.067,148.547
C03040=1204.101,148.104,-53.238,-178.174,6.069,148.547
C03041=1204.097,148.352,-53.259,-178.172,6.071,148.546
C03042=1204.092,148.601,-53.280,-178.170,6.072,148.546
C03043=1204.087,148.851,-53.301,-178.167,6.073,148.545
C03044=1204.083,149.100,-53.322,-178.164,6.075,148.545
C03045=1204.078,149.349,-53.343,-178.162,6.076,148.545
C03046=1204.073,149.598,-53.364,-178.159,6.077,148.544
C03047=1204.069,149.847,-53.385,-178.156,6.079,148.544
C03048=1204.064,150.096,-53.406,-178.154,6.080,148.543
C03049=1204.059,150.345,-53.427,-178.151,6.082,148.543
C03050=1204.055,150.594,-53.448,-178.148,6.083,148.542
C03051=1204.050,150.843,-53.469,-178.146,6.084,148.542
C03052=1204.045,151.093,-53.490,-178.143,6.086,148.541
C03053=1204.041,151.341,-53.511,-178.140,6.088,148.541
C03054=1204.035,151.590,-53.532,-178.138,6.088,148.540
C03055=1204.031,151.840,-53.554,-178.135,6.090,148.540
C03056=1204.027,152.088,-53.575,-178.133,6.092,148.540
C03057=1204.022,152.338,-53.596,-178.130,6.093,148.539
C03058=1204.017,152.586,-53.618,-178.127,6.094,148.539
C03059=1204.011,152.836,-53.638,-178.125,6.096,148.538
C03060=1204.008,153.085,-53.660,-178.122,6.098,148.538
C03061=1204.003,153.334,-53.681,-178.120,6.099,148.538
C03062=1203.998,153.583,-53.703,-178.117,6.101,148.537
C03063=1203.993,153.832,-53.724,-178.114,6.102,148.537
C03064=1203.989,154.081,-53.745,-178.112,6.103,148.536
C03065=1203.984,154.330,-53.766,-178.109,6.105,148.536
C03066=1203.979,154.579,-53.788,-178.107,6.107,148.535
C03067=1203.974,154.828,-53.809,-178.104,6.107,148.535
C03068=1203.970,155.077,-53.831,-178.101,6.109,148.534
C03069=1203.965,155.326,-53.851,-178.099,6.111,148.534
C03070=1203.960,155.575,-53.873,-178.096,6.112,148.534
C03071=1203.956,155.824,-53.894,-178.093,6.113,148.533
C03072=1203.951,156.074,-53.916,-178.091,6.115,148.533
C03073=1203.946,156.322,-53.937,-178.088,6.117,148.532
C03074=1203.941,156.571,-53.958,-178.086,6.118,148.532
C03075=1203.937,156.820,-53.980,-178.083,6.120,148.532
C03076=1203.933,157.069,-54.002,-178.080,6.121,148.531
C03077=1203.927,157.318,-54.022,-178.078,6.122,148.531
C03078=1203.923,157.568,-54.045,-178.075,6.124,148.530
C03079=1203.918,157.816,-54.066,-178.073,6.126,148.530
C03080=1203.913,158.066,-54.087,-178.069,6.127,148.529
C03081=1203.908,158.314,-54.109,-178.067,6.128,148.529
C03082=1203.904,158.564,-54.131,-178.065,6.130,148.529
C03083=1203.899,158.833,-54.154,-178.062,6.132,148.528
C03084=1203.894,159.102,-54.177,-178.059,6.133,148.528
C03085=1203.889,159.371,-54.200,-178.056,6.135,148.527
C03086=1203.884,159.640,-54.224,-178.053,6.137,148.527
C03087=1203.879,159.888,-54.246,-178.051,6.137,148.526
C03088=1203.874,160.138,-54.267,-178.048,6.139,148.526
C03089=1203.869,160.387,-54.289,-178.046,6.141,148.525
C03090=1203.865,160.636,-54.310,-178.043,6.143,148.525
C03091=1203.860,160.884,-54.332,-178.041,6.144,148.525
C03092=1203.855,161.134,-54.353,-178.038,6.145,148.524
C03093=1203.851,161.383,-54.374,-178.035,6.147,148.524
C03094=1203.847,161.632,-54.396,-178.032,6.149,148.523
C03095=1203.842,161.881,-54.418,-178.030,6.150,148.523
C03096=1203.837,162.129,-54.440,-178.027,6.152,148.523
C03097=1203.833,162.379,-54.462,-178.024,6.153,148.522
C03098=1203.828,162.628,-54.483,-178.022,6.155,148.522
C03099=1203.823,162.877,-54.505,-178.020,6.156,148.521
C03100=1203.818,163.126,-54.527,-178.017,6.158,148.521
C03101=1203.813,163.375,-54.549,-178.014,6.159,148.520
C03102=1203.809,163.624,-54.571,-178.012,6.161,148.520
C03103=1203.804,163.873,-54.593,-178.009,6.162,148.520
C03104=1203.799,164.122,-54.615,-178.006,6.164,148.519
C03105=1203.794,164.371,-54.636,-178.004,6.166,148.519
C03106=1203.790,164.620,-54.658,-178.001,6.167,148.518
C03107=1203.785,164.869,-54.680,-177.999,6.168,148.518
C03108=1203.780,165.117,-54.702,-177.996,6.170,148.518
C03109=1203.776,165.367,-54.724,-177.993,6.172,148.517
C03110=1203.771,165.615,-54.745,-177.990,6.173,148.517
C03111=1203.767,165.865,-54.767,-177.988,6.174,148.516
C03112=1203.762,166.113,-54.789,-177.986,6.176,148.516
C03113=1203.758,166.363,-54.811,-177.983,6.178,148.516
C03114=1203.752,166.612,-54.833,-177.980,6.180,148.515
C03115=1203.748,166.861,-54.856,-177.977,6.181,148.515
C03116=1203.743,167.110,-54.877,-177.975,6.182,148.514
C03117=1203.739,167.359,-54.899,-177.972,6.184,148.514
C03118=1203.734,167.608,-54.921,-177.970,6.186,148.514
C03119=1203.730,167.857,-54.943,-177.967,6.188,148.513
C03120=1203.724,168.106,-54.965,-177.965,6.189,148.513
C03121=1203.720,168.355,-54.987,-177.962,6.190,148.512
C03122=1203.715,168.604,-55.009,-177.959,6.192,148.512
C03123=1203.711,168.853,-55.031,-177.956,6.194,148.511
C03124=1203.706,169.101,-55.053,-177.954,6.195,148.511
C03125=1203.702,169.351,-55.075,-177.952,6.196,148.511
C03126=1203.696,169.599,-55.098,-177.949,6.198,148.510
C03127=1203.692,169.849,-55.120,-177.946,6.200,148.510
C03128=1203.687,170.097,-55.141,-177.944,6.202,148.510
C03129=1203.683,170.347,-55.164,-177.940,6.203,148.509
C03130=1203.678,170.595,-55.187,-177.938,6.204,148.509
C03131=1203.673,170.844,-55.209,-177.936,6.206,148.508
C03132=1203.669,171.093,-55.230,-177.933,6.208,148.508
C03133=1203.664,171.342,-55.252,-177.930,6.210,148.508
C03134=1203.659,171.591,-55.275,-177.928,6.211,148.507
C03135=1203.655,171.840,-55.297,-177.926,6.212,148.507
C03136=1203.650,172.089,-55.319,-177.923,6.214,148.506
C03137=1203.645,172.338,-55.342,-177.920,6.216,148.506
C03138=1203.641,172.588,-55.364,-177.917,6.217,148.505
C03139=1203.636,172.836,-55.386,-177.914,6.219,148.505
C03140=1203.632,173.085,-55.408,-177.912,6.220,148.505
C03141=1203.627,173.335,-55.431,-177.910,6.222,148.504
C03142=1203.622,173.583,-55.453,-177.907,6.224,148.504
C03143=1203.618,173.832,-55.475,-177.904,6.226,148.504
C03144=1203.612,174.081,-55.498,-177.902,6.227,148.503
C03145=1203.608,174.330,-55.520,-177.899,6.229,148.503
C03146=1203.603,174.579,-55.543,-177.896,6.230,148.502
C03147=1203.598,174.828,-55.565,-177.894,6.232,148.502
C03148=1203.594,175.077,-55.587,-177.891,6.234,148.502
C03149=1203.589,175.326,-55.610,-177.888,6.235,148.501
C03150=1203.585,175.575,-55.632,-177.886,6.237,148.501
C03151=1203.581,175.824,-55.654,-177.883,6.239,148.501
C03152=1203.575,176.072,-55.677,-177.881,6.240,148.500
C03153=1203.571,176.322,-55.700,-177.878,6.242,148.500
C03154=1203.566,176.571,-55.722,-177.876,6.244,148.499
C03155=1203.561,176.819,-55.745,-177.873,6.245,148.499
C03156=1203.557,177.069,-55.767,-177.870,6.247,148.499
C03157=1203.553,177.318,-55.790,-177.867,6.249,148.498
C03158=1203.548,177.566,-55.812,-177.865,6.250,148.498
C03159=1203.543,177.815,-55.835,-177.862,6.251,148.497
C03160=1203.539,178.065,-55.857,-177.860,6.253,148.497
C03161=1203.533,178.313,-55.880,-177.857,6.255,148.497
C03162=1203.529,178.562,-55.902,-177.854,6.257,148.496
C03163=1203.524,178.811,-55.925,-177.852,6.259,148.496
C03164=1203.520,179.059,-55.948,-177.849,6.260,148.496
C03165=1203.515,179.309,-55.970,-177.847,6.261,148.495
C03166=1203.511,179.558,-55.993,-177.844,6.263,148.495
C03167=1203.505,179.807,-56.016,-177.842,6.265,148.494
C03168=1203.501,180.055,-56.038,-177.839,6.267,148.494
C03169=1203.496,180.305,-56.061,-177.836,6.269,148.494
C03170=1203.492,180.554,-56.084,-177.833,6.270,148.493
C03171=1203.487,180.802,-56.107,-177.831,6.272,148.493
C03172=1203.483,181.051,-56.129,-177.829,6.273,148.492
C03173=1203.478,181.300,-56.152,-177.826,6.275,148.492
C03174=1203.474,181.549,-56.175,-177.823,6.277,148.492
C03175=1203.468,181.798,-56.197,-177.821,6.278,148.491
C03176=1203.465,182.047,-56.220,-177.818,6.280,148.491
C03177=1203.460,182.296,-56.243,-177.815,6.282,148.491
C03178=1203.455,182.546,-56.266,-177.813,6.284,148.490
C03179=1203.450,182.794,-56.288,-177.810,6.286,148.490
C03180=1203.446,183.043,-56.312,-177.808,6.287,148.490
C03181=1203.442,183.291,-56.334,-177.805,6.288,148.489
C03182=1203.437,183.541,-56.357,-177.802,6.290,148.489
C03183=1203.431,183.789,-56.380,-177.800,6.292,148.488
C03184=1203.427,184.038,-56.403,-177.797,6.294,148.488
C03185=1203.423,184.287,-56.426,-177.794,6.296,148.488
C03186=1203.418,184.536,-56.448,-177.792,6.297,148.487
C03187=1203.413,184.806,-56.474,-177.789,6.299,148.487
C03188=1203.408,185.075,-56.499,-177.786,6.301,148.486
C03189=1203.403,185.345,-56.523,-177.783,6.303,148.486
C03190=1203.398,185.614,-56.548,-177.781,6.304,148.486
C03191=1203.393,185.864,-56.572,-177.778,6.306,148.485
C03192=1203.389,186.112,-56.594,-177.775,6.308,148.485
C03193=1203.384,186.361,-56.617,-177.773,6.310,148.485
C03194=1203.379,186.610,-56.640,-177.770,6.312,148.484
C03195=1203.375,186.859,-56.663,-177.767,6.313,148.484
C03196=1203.371,187.108,-56.686,-177.765,6.315,148.484
C03197=1203.366,187.357,-56.710,-177.762,6.317,148.483
C03198=1203.361,187.606,-56.733,-177.759,6.319,148.483
C03199=1203.357,187.854,-56.755,-177.757,6.320,148.483
C03200=1203.352,188.103,-56.779,-177.755,6.322,148.482
C03201=1203.347,188.352,-56.802,-177.752,6.323,148.482
C03202=1203.342,188.601,-56.826,-177.749,6.325,148.482
C03203=1203.338,188.850,-56.848,-177.747,6.327,148.481
C03204=1203.334,189.099,-56.872,-177.744,6.329,148.481
C03205=1203.329,189.348,-56.895,-177.741,6.331,148.480
C03206=1203.324,189.596,-56.918,-177.739,6.333,148.480
C03207=1203.319,189.845,-56.941,-177.736,6.334,148.480
C03208=1203.315,190.094,-56.964,-177.733,6.336,148.479
C03209=1203.310,190.343,-56.988,-177.731,6.338,148.479
C03210=1203.306,190.592,-57.011,-177.728,6.340,148.479
C03211=1203.301,190.841,-57.034,-177.725,6.342,148.478
C03212=1203.296,191.090,-57.058,-177.723,6.343,148.478
C03213=1203.292,191.339,-57.081,-177.721,6.344,148.478
C03214=1203.288,191.588,-57.104,-177.718,6.346,148.477
C03215=1203.283,191.837,-57.127,-177.715,6.348,148.477
C03216=1203.278,192.086,-57.150,-177.713,6.350,148.477
C03217=1203.273,192.334,-57.174,-177.710,6.352,148.476
C03218=1203.269,192.583,-57.198,-177.707,6.353,148.476
C03219=1203.264,192.832,-57.221,-177.705,6.355,148.476
C03220=1203.259,193.081,-57.244,-177.702,6.357,148.475
C03221=1203.254,193.330,-57.268,-177.699,6.359,148.475
C03222=1203.251,193.579,-57.290,-177.697,6.361,148.475
C03223=1203.246,193.827,-57.314,-177.694,6.363,148.474
C03224=1203.241,194.076,-57.338,-177.692,6.364,148.474
C03225=1203.237,194.325,-57.361,-177.689,6.366,148.473
C03226=1203.232,194.574,-57.385,-177.686,6.368,148.473
C03227=1203.227,194.823,-57.408,-177.684,6.370,148.473
C03228=1203.223,195.071,-57.432,-177.681,6.372,148.472
C03229=1203.218,195.321,-57.455,-177.678,6.373,148.472
C03230=1203.214,195.570,-57.479,-177.676,6.375,148.472
C03231=1203.209,195.818,-57.503,-177.673,6.377,148.471
C03232=1203.204,196.067,-57.526,-177.670,6.379,148.471
C03233=1203.200,196.316,-57.549,-177.668,6.381,148.471
C03234=1203.195,196.565,-57.573,-177.665,6.383,148.470
C03235=1203.191,196.813,-57.597,-177.663,6.384,148.470
C03236=1203.186,197.063,-57.620,-177.660,6.385,148.470
C03237=1203.182,197.311,-57.644,-177.658,6.387,148.469
C03238=1203.177,197.560,-57.668,-177.655,6.389,148.469
C03239=1203.172,197.809,-57.691,-177.652,6.391,148.469
C03240=1203.168,198.057,-57.715,-177.650,6.393,148.468
C03241=1203.163,198.306,-57.738,-177.647,6.395,148.468
C03242=1203.158,198.555,-57.762,-177.645,6.397,148.468
C03243=1203.154,198.804,-57.786,-177.642,6.398,148.467
C03244=1203.149,199.053,-57.809,-177.640,6.400,148.467
C03245=1203.145,199.301,-57.833,-177.637,6.402,148.467
C03246=1203.141,199.551,-57.857,-177.634,6.404,148.466
C03247=1203.136,199.800,-57.882,-177.632,6.406,148.466
C03248=1203.131,200.049,-57.905,-177.629,6.408,148.466
C03249=1203.127,200.297,-57.929,-177.626,6.409,148.465
C03250=1203.122,200.546,-57.953,-177.624,6.411,148.465
C03251=1203.117,200.795,-57.977,-177.621,6.413,148.465
C03252=1203.113,201.044,-58.000,-177.618,6.415,148.464
C03253=1203.108,201.292,-58.024,-177.616,6.417,148.464
C03254=1203.104,201.541,-58.047,-177.613,6.418,148.464
C03255=1203.099,201.790,-58.072,-177.610,6.420,148.463
C03256=1203.094,202.040,-58.096,-177.608,6.422,148.463
C03257=1203.090,202.288,-58.120,-177.606,6.424,148.463
C03258=1203.085,202.537,-58.143,-177.603,6.426,148.462
C03259=1203.081,202.785,-58.167,-177.600,6.428,148.462
C03260=1203.077,203.034,-58.191,-177.598,6.430,148.462
C03261=1203.071,203.283,-58.215,-177.595,6.432,148.461
C03262=1203.067,203.532,-58.239,-177.592,6.433,148.461
C03263=1203.062,203.780,-58.263,-177.590,6.435,148.461
C03264=1203.058,204.030,-58.287,-177.587,6.437,148.460
C03265=1203.054,204.278,-58.311,-177.584,6.439,148.460
C03266=1203.049,204.527,-58.336,-177.581,6.442,148.460
C03267=1203.044,204.776,-58.359,-177.579,6.444,148.460
C03268=1203.040,205.024,-58.383,-177.576,6.445,148.459
C03269=1203.035,205.273,-58.407,-177.574,6.447,148.459
C03270=1203.030,205.523,-58.432,-177.571,6.449,148.459
C03271=1203.026,205.771,-58.456,-177.568,6.451,148.458
C03272=1203.022,206.020,-58.480,-177.566,6.453,148.458
C03273=1203.017,206.268,-58.504,-177.563,6.455,148.458
C03274=1203.012,206.517,-58.528,-177.560,6.456,148.457
C03275=1203.008,206.767,-58.552,-177.558,6.458,148.457
C03276=1203.004,207.015,-58.576,-177.556,6.460,148.457
C03277=1202.998,207.264,-58.601,-177.553,6.462,148.456
C03278=1202.994,207.513,-58.624,-177.550,6.464,148.456
C03279=1202.989,207.761,-58.649,-177.548,6.466,148.456
C03280=1202.985,208.011,-58.674,-177.545,6.468,148.455
C03281=1202.980,208.259,-58.698,-177.542,6.470,148.455
C03282=1202.976,208.507,-58.722,-177.540,6.471,148.455
C03283=1202.971,208.756,-58.746,-177.537,6.473,148.454
C03284=1202.967,209.005,-58.771,-177.535,6.475,148.454
C03285=1202.962,209.255,-58.795,-177.532,6.477,148.454
C03286=1202.957,209.503,-58.819,-177.530,6.479,148.454
C03287=1202.953,209.751,-58.843,-177.527,6.481,148.453
C03288=1202.948,210.001,-58.868,-177.524,6.483,148.453
C03289=1202.944,210.249,-58.892,-177.521,6.485,148.453
C03290=1202.939,210.498,-58.917,-177.518,6.487,148.452
C03291=1202.934,210.768,-58.943,-177.516,6.489,148.452
C03292=1202.930,211.039,-58.970,-177.513,6.491,148.452
C03293=1202.924,211.309,-58.996,-177.510,6.493,148.451
C03294=1202.919,211.580,-59.023,-177.507,6.495,148.451
C03295=1202.915,211.828,-59.047,-177.505,6.497,148.451
C03296=1202.910,212.077,-59.072,-177.502,6.499,148.451
C03297=1202.906,212.326,-59.096,-177.500,6.501,148.450
C03298=1202.901,212.575,-59.120,-177.497,6.503,148.450
C03299=1202.897,212.824,-59.145,-177.495,6.505,148.450
C03300=1202.892,213.072,-59.170,-177.491,6.507,148.449
C03301=1202.887,213.321,-59.194,-177.489,6.509,148.449
C03302=1202.883,213.570,-59.219,-177.486,6.511,148.449
C03303=1202.879,213.818,-59.243,-177.484,6.513,148.448
C03304=1202.874,214.067,-59.268,-177.481,6.515,148.448
C03305=1202.870,214.316,-59.293,-177.479,6.517,148.448
C03306=1202.865,214.565,-59.317,-177.476,6.519,148.447
C03307=1202.860,214.813,-59.341,-177.473,6.521,148.447
C03308=1202.856,215.062,-59.366,-177.471,6.522,148.447
C03309=1202.851,215.311,-59.390,-177.469,6.525,148.447
C03310=1202.846,215.560,-59.415,-177.466,6.526,148.446
C03311=1202.843,215.808,-59.440,-177.463,6.529,148.446
C03312=1202.838,216.057,-59.465,-177.460,6.531,148.446
C03313=1202.833,216.306,-59.490,-177.457,6.533,148.445
C03314=1202.829,216.555,-59.514,-177.455,6.535,148.445
C03315=1202.824,216.803,-59.539,-177.453,6.537,148.445
C03316=1202.820,217.052,-59.564,-177.450,6.539,148.445
C03317=1202.815,217.301,-59.589,-177.447,6.540,148.444
C03318=1202.810,217.549,-59.613,-177.445,6.542,148.444
C03319=1202.806,217.798,-59.638,-177.442,6.544,148.444
C03320=1202.801,218.046,-59.663,-177.439,6.547,148.444
C03321=1202.797,218.296,-59.688,-177.437,6.549,148.443
C03322=1202.792,218.544,-59.712,-177.434,6.551,148.443
C03323=1202.788,218.793,-59.738,-177.431,6.552,148.443
C03324=1202.783,219.042,-59.763,-177.429,6.554,148.442
C03325=1202.779,219.290,-59.787,-177.427,6.556,148.442
C03326=1202.774,219.539,-59.812,-177.424,6.558,148.442
C03327=1202.769,219.788,-59.837,-177.421,6.560,148.441
C03328=1202.765,220.037,-59.862,-177.419,6.562,148.441
C03329=1202.761,220.285,-59.887,-177.415,6.565,148.441
C03330=1202.756,220.534,-59.912,-177.413,6.567,148.441
C03331=1202.752,220.782,-59.937,-177.411,6.569,148.440
C03332=1202.747,221.032,-59.962,-177.408,6.570,148.440
C03333=1202.742,221.280,-59.986,-177.405,6.572,148.440
C03334=1202.738,221.529,-60.012,-177.403,6.574,148.440
C03335=1202.734,221.778,-60.036,-177.401,6.576,148.439
C03336=1202.730,222.026,-60.062,-177.398,6.578,148.439
C03337=1202.724,222.275,-60.087,-177.395,6.581,148.439
C03338=1202.720,222.524,-60.112,-177.393,6.583,148.439
C03339=1202.716,222.772,-60.137,-177.390,6.585,148.438
C03340=1202.712,223.021,-60.162,-177.387,6.587,148.438
C03341=1202.706,223.270,-60.187,-177.385,6.588,148.438
C03342=1202.702,223.519,-60.213,-177.382,6.590,148.437
C03343=1202.697,223.767,-60.237,-177.380,6.592,148.437
C03344=1202.694,224.016,-60.262,-177.377,6.595,148.437
C03345=1202.689,224.264,-60.288,-177.374,6.597,148.437
C03346=1202.684,224.513,-60.313,-177.371,6.599,148.436
C03347=1202.679,224.762,-60.338,-177.369,6.601,148.436
C03348=1202.675,225.011,-60.363,-177.367,6.603,148.436
C03349=1202.670,225.259,-60.389,-177.364,6.605,148.435
C03350=1202.666,225.508,-60.414,-177.361,6.606,148.435
C03351=1202.661,225.756,-60.439,-177.359,6.609,148.435
C03352=1202.657,226.005,-60.464,-177.356,6.611,148.435
C03353=1202.653,226.255,-60.489,-177.353,6.613,148.434
C03354=1202.648,226.503,-60.515,-177.351,6.615,148.434
C03355=1202.644,226.751,-60.540,-177.348,6.617,148.434
C03356=1202.639,227.000,-60.566,-177.346,6.619,148.434
C03357=1202.634,227.249,-60.591,-177.343,6.622,148.433
C03358=1202.629,227.497,-60.616,-177.340,6.624,148.433
C03359=1202.625,227.746,-60.642,-177.338,6.626,148.433
C03360=1202.621,227.995,-60.667,-177.335,6.627,148.433
C03361=1202.616,228.243,-60.692,-177.333,6.629,148.432
C03362=1202.612,228.492,-60.718,-177.330,6.631,148.432
C03363=1202.607,228.741,-60.744,-177.327,6.634,148.432
C03364=1202.603,228.989,-60.768,-177.325,6.636,148.432
C03365=1202.599,229.238,-60.794,-177.322,6.638,148.431
C03366=1202.594,229.486,-60.819,-177.320,6.640,148.431
C03367=1202.590,229.735,-60.845,-177.317,6.642,148.431
C03368=1202.585,229.984,-60.871,-177.315,6.644,148.431
C03369=1202.581,230.232,-60.896,-177.312,6.647,148.430
C03370=1202.576,230.481,-60.921,-177.309,6.648,148.430
C03371=1202.572,230.730,-60.947,-177.306,6.650,148.430
C03372=1202.566,230.979,-60.973,-177.304,6.652,148.430
C03373=1202.562,231.227,-60.999,-177.302,6.654,148.429
C03374=1202.558,231.476,-61.024,-177.299,6.656,148.429
C03375=1202.553,231.724,-61.050,-177.296,6.659,148.429
C03376=1202.549,231.973,-61.075,-177.294,6.661,148.429
C03377=1202.545,232.222,-61.101,-177.291,6.663,148.428
C03378=1202.540,232.470,-61.127,-177.289,6.665,148.428
C03379=1202.536,232.719,-61.152,-177.286,6.667,148.428
C03380=1202.531,232.968,-61.178,-177.283,6.670,148.428
C03381=1202.526,233.216,-61.203,-177.281,6.672,148.427
C03382=1202.522,233.465,-61.229,-177.278,6.674,148.427
C03383=1202.518,233.714,-61.254,-177.276,6.675,148.427
C03384=1202.512,233.962,-61.280,-177.273,6.678,148.427
C03385=1202.508,234.211,-61.307,-177.270,6.680,148.426
C03386=1202.504,234.459,-61.332,-177.268,6.682,148.426
C03387=1202.500,234.708,-61.358,-177.266,6.684,148.426
C03388=1202.495,234.956,-61.384,-177.263,6.686,148.426
C03389=1202.491,235.205,-61.409,-177.260,6.688,148.425
C03390=1202.487,235.454,-61.435,-177.258,6.691,148.425
C03391=1202.482,235.703,-61.461,-177.255,6.693,148.425
C03392=1202.477,235.951,-61.487,-177.252,6.695,148.425
C03393=1202.473,236.200,-61.513,-177.250,6.697,148.425
C03394=1202.468,236.449,-61.538,-177.247,6.699,148.424
C03395=1202.463,236.719,-61.567,-177.244,6.701,148.424
C03396=1202.459,236.991,-61.595,-177.242,6.703,148.424
C03397=1202.453,237.263,-61.623,-177.239,6.706,148.424
C03398=1202.448,237.534,-61.652,-177.236,6.708,148.423
C03399=1202.444,237.783,-61.678,-177.233,6.711,148.423
C03400=1202.440,238.032,-61.703,-177.231,6.713,148.423
C03401=1202.435,238.281,-61.730,-177.228,6.715,148.423
C03402=1202.431,238.529,-61.756,-177.226,6.716,148.422
C03403=1202.426,238.777,-61.781,-177.223,6.719,148.422
C03404=1202.422,239.026,-61.807,-177.220,6.721,148.422
C03405=1202.417,239.275,-61.834,-177.218,6.723,148.422
C03406=1202.413,239.523,-61.860,-177.216,6.725,148.421
C03407=1202.409,239.772,-61.886,-177.213,6.727,148.421
C03408=1202.404,240.021,-61.912,-177.210,6.730,148.421
C03409=1202.399,240.269,-61.938,-177.208,6.732,148.421
C03410=1202.395,240.517,-61.964,-177.205,6.734,148.421
C03411=1202.390,240.767,-61.990,-177.203,6.736,148.420
C03412=1202.386,241.015,-62.017,-177.200,6.739,148.420
C03413=1202.382,241.263,-62.043,-177.197,6.741,148.420
C03414=1202.377,241.513,-62.069,-177.195,6.743,148.420
C03415=1202.372,241.760,-62.095,-177.193,6.745,148.420
C03416=1202.368,242.009,-62.121,-177.189,6.748,148.419
C03417=1202.363,242.258,-62.147,-177.187,6.749,148.419
C03418=1202.359,242.506,-62.174,-177.185,6.752,148.419
C03419=1202.355,242.755,-62.199,-177.182,6.753,148.418
C03420=1202.350,243.003,-62.226,-177.179,6.756,148.418
C03421=1202.346,243.252,-62.252,-177.177,6.758,148.418
C03422=1202.342,243.501,-62.279,-177.174,6.760,148.418
C03423=1202.337,243.749,-62.305,-177.172,6.762,148.418
C03424=1202.332,243.998,-62.331,-177.169,6.765,148.417
C03425=1202.328,244.246,-62.357,-177.167,6.767,148.417
C03426=1202.324,244.495,-62.383,-177.164,6.769,148.417
C03427=1202.319,244.743,-62.410,-177.162,6.771,148.417
C03428=1202.315,244.992,-62.437,-177.159,6.774,148.417
C03429=1202.310,245.241,-62.463,-177.156,6.776,148.416
C03430=1202.306,245.489,-62.489,-177.154,6.778,148.416
C03431=1202.301,245.738,-62.516,-177.151,6.781,148.416
C03432=1202.297,245.986,-62.542,-177.148,6.783,148.416
C03433=1202.292,246.235,-62.569,-177.146,6.785,148.416
C03434=1202.288,246.484,-62.595,-177.144,6.787,148.415
C03435=1202.284,246.732,-62.622,-177.140,6.789,148.415
C03436=1202.280,246.981,-62.648,-177.138,6.792,148.415
C03437=1202.275,247.229,-62.675,-177.136,6.793,148.415
C03438=1202.270,247.477,-62.700,-177.133,6.795,148.414
C03439=1202.265,247.726,-62.727,-177.130,6.798,148.414
C03440=1202.261,247.974,-62.754,-177.128,6.800,148.414
C03441=1202.257,248.223,-62.780,-177.126,6.802,148.414
C03442=1202.252,248.472,-62.807,-177.122,6.805,148.414
C03443=1202.248,248.720,-62.834,-177.120,6.807,148.414
C03444=1202.243,248.968,-62.861,-177.118,6.809,148.413
C03445=1202.239,249.217,-62.887,-177.115,6.812,148.413
C03446=1202.234,249.466,-62.914,-177.112,6.814,148.413
C03447=1202.230,249.714,-62.941,-177.110,6.816,148.413
C03448=1202.226,249.963,-62.966,-177.108,6.818,148.413
C03449=1202.221,250.212,-62.994,-177.105,6.821,148.413
C03450=1202.217,250.460,-63.020,-177.102,6.823,148.412
C03451=1202.212,250.708,-63.047,-177.100,6.825,148.412
C03452=1202.208,250.957,-63.074,-177.097,6.828,148.412
C03453=1202.204,251.206,-63.100,-177.095,6.830,148.412
C03454=1202.199,251.455,-63.127,-177.092,6.832,148.411
C03455=1202.195,251.703,-63.154,-177.089,6.835,148.411
C03456=1202.191,251.951,-63.181,-177.087,6.836,148.411
C03457=1202.186,252.200,-63.208,-177.085,6.839,148.411
C03458=1202.181,252.448,-63.235,-177.081,6.841,148.411
C03459=1202.177,252.697,-63.262,-177.079,6.843,148.411
C03460=1202.173,252.945,-63.288,-177.077,6.845,148.410
C03461=1202.168,253.194,-63.315,-177.074,6.847,148.410
C03462=1202.163,253.443,-63.342,-177.071,6.850,148.410
C03463=1202.159,253.691,-63.368,-177.069,6.852,148.410
C03464=1202.155,253.939,-63.395,-177.067,6.854,148.410
C03465=1202.150,254.188,-63.422,-177.064,6.857,148.409
C03466=1202.145,254.436,-63.450,-177.061,6.859,148.409
C03467=1202.142,254.685,-63.476,-177.059,6.861,148.409
C03468=1202.137,254.934,-63.503,-177.056,6.864,148.409
C03469=1202.133,255.182,-63.530,-177.054,6.866,148.409
C03470=1202.128,255.431,-63.558,-177.051,6.868,148.408
C03471=1202.123,255.679,-63.585,-177.048,6.871,148.408
C03472=1202.120,255.927,-63.611,-177.046,6.873,148.408
C03473=1202.115,256.176,-63.638,-177.044,6.875,148.408
C03474=1202.110,256.424,-63.665,-177.040,6.878,148.408
C03475=1202.106,256.674,-63.693,-177.038,6.880,148.408
C03476=1202.102,256.921,-63.720,-177.035,6.883,148.407
C03477=1202.098,257.170,-63.747,-177.033,6.885,148.407
C03478=1202.093,257.418,-63.774,-177.030,6.887,148.407
C03479=1202.089,257.667,-63.801,-177.028,6.890,148.407
C03480=1202.084,257.915,-63.828,-177.025,6.892,148.407
C03481=1202.079,258.164,-63.855,-177.023,6.894,148.407
C03482=1202.075,258.413,-63.883,-177.020,6.897,148.406
C03483=1202.071,258.661,-63.910,-177.017,6.898,148.406
C03484=1202.066,258.909,-63.937,-177.015,6.901,148.406
C03485=1202.062,259.157,-63.964,-177.012,6.903,148.406
C03486=1202.058,259.406,-63.991,-177.010,6.905,148.406
C03487=1202.054,259.655,-64.018,-177.007,6.907,148.405
C03488=1202.049,259.904,-64.045,-177.005,6.910,148.405
C03489=1202.045,260.151,-64.073,-177.003,6.913,148.405
C03490=1202.040,260.400,-64.100,-176.999,6.915,148.405
C03491=1202.035,260.648,-64.127,-176.997,6.917,148.405
C03492=1202.031,260.897,-64.155,-176.995,6.919,148.405
C03493=1202.027,261.146,-64.182,-176.992,6.922,148.405
C03494=1202.022,261.394,-64.210,-176.989,6.924,148.404
C03495=1202.018,261.643,-64.237,-176.987,6.927,148.404
C03496=1202.014,261.891,-64.265,-176.984,6.929,148.404
C03497=1202.009,262.140,-64.292,-176.982,6.931,148.404
C03498=1202.004,262.388,-64.319,-176.979,6.934,148.404
C03499=1201.999,262.661,-64.349,-176.976,6.936,148.404
C03500=1201.995,262.934,-64.379,-176.974,6.939,148.403
C03501=1201.990,263.206,-64.410,-176.971,6.942,148.403
C03502=1201.985,263.479,-64.439,-176.968,6.945,148.403
C03503=1201.982,263.727,-64.467,-176.965,6.947,148.403
C03504=1201.977,263.976,-64.494,-176.963,6.949,148.403
C03505=1201.972,264.225,-64.522,-176.960,6.951,148.403
C03506=1201.967,264.472,-64.550,-176.958,6.954,148.402
C03507=1201.963,264.722,-64.577,-176.955,6.957,148.402
C03508=1201.959,264.969,-64.605,-176.952,6.958,148.402
C03509=1201.954,265.218,-64.632,-176.950,6.961,148.402
C03510=1201.950,265.467,-64.660,-176.948,6.964,148.402
C03511=1201.946,265.715,-64.687,-176.945,6.966,148.402
C03512=1201.941,265.963,-64.715,-176.942,6.969,148.402
C03513=1201.937,266.212,-64.743,-176.940,6.970,148.401
C03514=1201.932,266.460,-64.771,-176.938,6.973,148.401
C03515=1201.928,266.709,-64.798,-176.935,6.976,148.401
C03516=1201.924,266.957,-64.826,-176.932,6.977,148.401
C03517=1201.920,267.205,-64.854,-176.929,6.980,148.401
C03518=1201.915,267.454,-64.881,-176.927,6.983,148.401
C03519=1201.911,267.702,-64.909,-176.924,6.985,148.401
C03520=1201.906,267.951,-64.937,-176.922,6.987,148.400
C03521=1201.901,268.199,-64.965,-176.920,6.990,148.400
C03522=1201.898,268.448,-64.993,-176.917,6.992,148.400
C03523=1201.893,268.696,-65.020,-176.915,6.995,148.400
C03524=1201.889,268.944,-65.048,-176.911,6.997,148.400
C03525=1201.884,269.193,-65.076,-176.909,6.999,148.400
C03526=1201.880,269.441,-65.103,-176.907,7.002,148.400
C03527=1201.876,269.690,-65.132,-176.904,7.004,148.399
C03528=1201.871,269.938,-65.159,-176.902,7.006,148.399
C03529=1201.866,270.187,-65.187,-176.899,7.009,148.399
C03530=1201.862,270.435,-65.215,-176.896,7.011,148.399
C03531=1201.858,270.683,-65.243,-176.894,7.014,148.399
C03532=1201.854,270.932,-65.271,-176.892,7.017,148.399
C03533=1201.849,271.180,-65.299,-176.888,7.019,148.399
C03534=1201.844,271.428,-65.326,-176.886,7.021,148.398
C03535=1201.841,271.677,-65.355,-176.884,7.024,148.398
C03536=1201.836,271.925,-65.383,-176.881,7.027,148.398
C03537=1201.832,272.174,-65.411,-176.879,7.028,148.398
C03538=1201.828,272.422,-65.439,-176.876,7.031,148.398
C03539=1201.823,272.671,-65.466,-176.874,7.034,148.398
C03540=1201.818,272.919,-65.495,-176.871,7.036,148.398
C03541=1201.815,273.167,-65.523,-176.869,7.039,148.398
C03542=1201.810,273.416,-65.551,-176.866,7.042,148.398
C03543=1201.805,273.664,-65.579,-176.863,7.043,148.397
C03544=1201.801,273.912,-65.607,-176.861,7.046,148.397
C03545=1201.796,274.160,-65.635,-176.858,7.049,148.397
C03546=1201.793,274.409,-65.664,-176.855,7.051,148.397
C03547=1201.788,274.657,-65.691,-176.853,7.053,148.397
C03548=1201.784,274.906,-65.720,-176.850,7.056,148.397
C03549=1201.779,275.154,-65.748,-176.848,7.059,148.397
C03550=1201.775,275.402,-65.777,-176.845,7.061,148.396
C03551=1201.771,275.650,-65.804,-176.843,7.064,148.396
C03552=1201.767,275.899,-65.833,-176.840,7.067,148.396
C03553=1201.762,276.147,-65.861,-176.838,7.069,148.396
C03554=1201.758,276.396,-65.889,-176.836,7.071,148.396
C03555=1201.753,276.644,-65.917,-176.833,7.074,148.396
C03556=1201.749,276.892,-65.946,-176.831,7.076,148.396
C03557=1201.745,277.141,-65.974,-176.828,7.078,148.396
C03558=1201.740,277.389,-66.002,-176.825,7.081,148.396
C03559=1201.736,277.638,-66.031,-176.823,7.084,148.396
C03560=1201.731,277.886,-66.059,-176.821,7.086,148.395
C03561=1201.727,278.135,-66.087,-176.817,7.089,148.395
C03562=1201.723,278.383,-66.115,-176.815,7.091,148.395
C03563=1201.718,278.632,-66.144,-176.813,7.094,148.395
C03564=1201.714,278.879,-66.172,-176.810,7.096,148.395
C03565=1201.710,279.128,-66.201,-176.807,7.099,148.395
C03566=1201.706,279.376,-66.229,-176.805,7.101,148.395
C03567=1201.701,279.624,-66.258,-176.802,7.104,148.395
C03568=1201.697,279.873,-66.286,-176.800,7.106,148.395
C03569=1201.692,280.121,-66.315,-176.797,7.109,148.394
C03570=1201.688,280.370,-66.344,-176.795,7.111,148.394
C03571=1201.684,280.618,-66.372,-176.792,7.114,148.394
C03572=1201.679,280.866,-66.400,-176.790,7.116,148.394
C03573=1201.675,281.115,-66.428,-176.787,7.119,148.394
C03574=1201.670,281.362,-66.457,-176.784,7.122,148.394
C03575=1201.666,281.611,-66.486,-176.782,7.124,148.394
C03576=1201.662,281.860,-66.514,-176.779,7.127,148.394
C03577=1201.657,282.107,-66.543,-176.777,7.129,148.394
C03578=1201.654,282.356,-66.571,-176.775,7.132,148.394
C03579=1201.649,282.605,-66.600,-176.772,7.134,148.393
C03580=1201.644,282.852,-66.629,-176.769,7.137,148.393
C03581=1201.641,283.101,-66.657,-176.767,7.139,148.393
C03582=1201.635,283.349,-66.686,-176.764,7.142,148.393
C03583=1201.631,283.597,-66.715,-176.762,7.144,148.393
C03584=1201.628,283.846,-66.743,-176.759,7.147,148.393
C03585=1201.623,284.094,-66.772,-176.757,7.149,148.393
C03586=1201.618,284.343,-66.801,-176.754,7.152,148.393
C03587=1201.614,284.591,-66.830,-176.752,7.155,148.393
C03588=1201.610,284.839,-66.858,-176.749,7.158,148.393
C03589=1201.605,285.088,-66.887,-176.747,7.159,148.392
C03590=1201.601,285.336,-66.917,-176.744,7.162,148.392
C03591=1201.597,285.585,-66.945,-176.741,7.165,148.392
C03592=1201.593,285.832,-66.974,-176.739,7.168,148.392
C03593=1201.588,286.081,-67.003,-176.737,7.171,148.392
C03594=1201.584,286.329,-67.032,-176.734,7.173,148.392
C03595=1201.579,286.577,-67.060,-176.731,7.176,148.392
C03596=1201.575,286.825,-67.089,-176.729,7.178,148.392
C03597=1201.571,287.074,-67.118,-176.726,7.181,148.392
C03598=1201.567,287.322,-67.147,-176.724,7.183,148.392
C03599=1201.562,287.570,-67.177,-176.722,7.186,148.392
C03600=1201.557,287.819,-67.205,-176.719,7.188,148.392
C03601=1201.554,288.067,-67.234,-176.716,7.191,148.391
C03602=1201.549,288.316,-67.263,-176.714,7.194,148.391
C03603=1201.545,288.589,-67.295,-176.711,7.197,148.391
C03604=1201.539,288.864,-67.327,-176.709,7.199,148.391
C03605=1201.535,289.138,-67.359,-176.706,7.202,148.391
C03606=1201.530,289.412,-67.391,-176.703,7.205,148.391
C03607=1201.526,289.661,-67.420,-176.700,7.208,148.391
C03608=1201.521,289.909,-67.450,-176.698,7.210,148.391
C03609=1201.517,290.158,-67.479,-176.695,7.213,148.391
C03610=1201.512,290.406,-67.508,-176.693,7.216,148.391
C03611=1201.508,290.654,-67.537,-176.691,7.218,148.391
C03612=1201.504,290.902,-67.566,-176.688,7.221,148.391
C03613=1201.500,291.150,-67.595,-176.686,7.223,148.391
C03614=1201.496,291.399,-67.624,-176.683,7.226,148.391
C03615=1201.491,291.647,-67.653,-176.680,7.228,148.390
C03616=1201.487,291.895,-67.683,-176.678,7.231,148.390
C03617=1201.483,292.143,-67.712,-176.675,7.234,148.390
C03618=1201.479,292.392,-67.741,-176.673,7.236,148.390
C03619=1201.474,292.640,-67.770,-176.670,7.240,148.390
C03620=1201.470,292.889,-67.800,-176.668,7.242,148.390
C03621=1201.465,293.136,-67.829,-176.665,7.245,148.390
C03622=1201.461,293.385,-67.858,-176.663,7.248,148.390
C03623=1201.457,293.633,-67.888,-176.660,7.250,148.390
C03624=1201.453,293.881,-67.917,-176.658,7.253,148.390
C03625=1201.448,294.129,-67.947,-176.655,7.255,148.390
C03626=1201.444,294.378,-67.976,-176.652,7.258,148.390
C03627=1201.440,294.626,-68.005,-176.650,7.261,148.390
C03628=1201.435,294.874,-68.034,-176.648,7.263,148.390
C03629=1201.431,295.122,-68.063,-176.645,7.266,148.390
C03630=1201.427,295.371,-68.093,-176.643,7.268,148.390
C03631=1201.422,295.619,-68.122,-176.640,7.271,148.390
C03632=1201.418,295.867,-68.152,-176.638,7.273,148.390
C03633=1201.414,296.115,-68.181,-176.635,7.276,148.390
C03634=1201.409,296.364,-68.211,-176.633,7.279,148.390
C03635=1201.405,296.612,-68.241,-176.630,7.282,148.389
C03636=1201.401,296.861,-68.270,-176.628,7.285,148.389
C03637=1201.397,297.108,-68.300,-176.625,7.288,148.389
C03638=1201.393,297.356,-68.330,-176.623,7.290,148.389
C03639=1201.389,297.605,-68.359,-176.620,7.293,148.389
C03640=1201.384,297.852,-68.388,-176.618,7.295,148.389
C03641=1201.380,298.101,-68.418,-176.615,7.298,148.389
C03642=1201.375,298.349,-68.448,-176.613,7.301,148.389
C03643=1201.370,298.597,-68.477,-176.611,7.303,148.389
C03644=1201.366,298.846,-68.507,-176.608,7.306,148.389
C03645=1201.362,299.094,-68.536,-176.606,7.309,148.389
C03646=1201.358,299.342,-68.566,-176.603,7.312,148.389
C03647=1201.354,299.590,-68.596,-176.600,7.315,148.389
C03648=1201.349,299.838,-68.626,-176.598,7.317,148.389
C03649=1201.345,300.087,-68.655,-176.596,7.320,148.389
C03650=1201.341,300.335,-68.685,-176.593,7.322,148.389
C03651=1201.337,300.583,-68.715,-176.591,7.325,148.389
C03652=1201.332,300.831,-68.745,-176.588,7.328,148.389
C03653=1201.328,301.079,-68.774,-176.586,7.330,148.389
C03654=1201.324,301.328,-68.804,-176.583,7.333,148.389
C03655=1201.320,301.575,-68.834,-176.581,7.336,148.389
